//
FOR _i := GVL.PROG_CMDS_ARR_BEG TO GVL.PROG_CMDS_ARR_END BY 1 DO
	PersistentVars.Programs[11].Commands[_i].CommandType := DUT_CommandType.Disabled;
	PersistentVars.Programs[11].Commands[_i].CommandString := '';
END_FOR
PersistentVars.Programs[11].ProgramName := 'Make Me an Egg, Please';
PersistentVars.Programs[11].Commands[0].CommandType := DUT_CommandType.Disabled;
PersistentVars.Programs[11].Commands[0].CommandString := '';

//
FOR _i := GVL.PROG_CMDS_ARR_BEG TO GVL.PROG_CMDS_ARR_END BY 1 DO
	PersistentVars.Programs[12].Commands[_i].CommandType := DUT_CommandType.Disabled;
	PersistentVars.Programs[12].Commands[_i].CommandString := '';
END_FOR
PersistentVars.Programs[12].ProgramName := 'Egg Pick Routine';
PersistentVars.Programs[12].Commands[0].CommandType := DUT_CommandType.Disabled;
PersistentVars.Programs[12].Commands[0].CommandString := '';

//
FOR _i := GVL.PROG_CMDS_ARR_BEG TO GVL.PROG_CMDS_ARR_END BY 1 DO
	PersistentVars.Programs[13].Commands[_i].CommandType := DUT_CommandType.Disabled;
	PersistentVars.Programs[13].Commands[_i].CommandString := '';
END_FOR
PersistentVars.Programs[13].ProgramName := 'Egg Crack Routine';
PersistentVars.Programs[13].Commands[0].CommandType := DUT_CommandType.Disabled;
PersistentVars.Programs[13].Commands[0].CommandString := '';

//
FOR _i := GVL.PROG_CMDS_ARR_BEG TO GVL.PROG_CMDS_ARR_END BY 1 DO
	PersistentVars.Programs[14].Commands[_i].CommandType := DUT_CommandType.Disabled;
	PersistentVars.Programs[14].Commands[_i].CommandString := '';
END_FOR
PersistentVars.Programs[14].ProgramName := 'Egg Flip Routine';
PersistentVars.Programs[14].Commands[0].CommandType := DUT_CommandType.Disabled;
PersistentVars.Programs[14].Commands[0].CommandString := '';

//
FOR _i := GVL.PROG_CMDS_ARR_BEG TO GVL.PROG_CMDS_ARR_END BY 1 DO
	PersistentVars.Programs[15].Commands[_i].CommandType := DUT_CommandType.Disabled;
	PersistentVars.Programs[15].Commands[_i].CommandString := '';
END_FOR
PersistentVars.Programs[15].ProgramName := 'Egg Place Routine';
PersistentVars.Programs[15].Commands[0].CommandType := DUT_CommandType.Disabled;
PersistentVars.Programs[15].Commands[0].CommandString := '';
END_METHOD

METHOD M_Init : BOOL

// check if arfbot has been initialized
IF NOT PersistentVars.Flags[GVL.INIT_POS_IDX].Value THEN
	// poses
	PersistentVars.Flags[GVL.HOM_TO_POSE_IDX].Value := FALSE;
	PersistentVars.StoredPositions[GVL.POSE_1_IDX].Position.X := 0.0;
	PersistentVars.StoredPositions[GVL.POSE_1_IDX].Position.Y := -15.0;
	PersistentVars.StoredPositions[GVL.POSE_1_IDX].Position.Z := 115.0;
	PersistentVars.StoredPositions[GVL.POSE_1_IDX].Position.A := 0.0;
	PersistentVars.StoredPositions[GVL.POSE_1_IDX].Position.B := 30.0;
	PersistentVars.StoredPositions[GVL.POSE_1_IDX].Position.C := 0.0;
	
	PersistentVars.StoredPositions[GVL.POSE_2_IDX].Position.X := 0.0;
	PersistentVars.StoredPositions[GVL.POSE_2_IDX].Position.Y := -15.0;
	PersistentVars.StoredPositions[GVL.POSE_2_IDX].Position.Z := 115.0;
	PersistentVars.StoredPositions[GVL.POSE_2_IDX].Position.A := 0.0;
	PersistentVars.StoredPositions[GVL.POSE_2_IDX].Position.B := -30.0;
	PersistentVars.StoredPositions[GVL.POSE_2_IDX].Position.C := 0.0;
		 
	// decoder
	PersistentVars.StoredPositions[GVL.DEC_START_POS].Position.X := 300.0; // TODO need to verify all 6 of these
	PersistentVars.StoredPositions[GVL.DEC_START_POS].Position.Y := 0.0;
	PersistentVars.StoredPositions[GVL.DEC_START_POS].Position.Z := -400.0;
	PersistentVars.StoredPositions[GVL.DEC_START_POS].Position.A := 0.0;
	PersistentVars.StoredPositions[GVL.DEC_START_POS].Position.B := 0.0;
	PersistentVars.StoredPositions[GVL.DEC_START_POS].Position.C := 0.0;
	
	// set homing offsets
	PersistentVars.StoredPositions[GVL.HOM_POS_IDX].Position.X := 166; // J1 initial home offset
	PersistentVars.StoredPositions[GVL.HOM_POS_IDX].Position.Y := -35.3; // J2 initial home offset
	PersistentVars.StoredPositions[GVL.HOM_POS_IDX].Position.Z := 145; // J3 initial home offset
	PersistentVars.StoredPositions[GVL.HOM_POS_IDX].Position.A := -166; // J4 initial home offset
	PersistentVars.StoredPositions[GVL.HOM_POS_IDX].Position.B := -99.2; // J5 initial home offset
	PersistentVars.StoredPositions[GVL.HOM_POS_IDX].Position.C := 178; // J6 initial home offset
	
	// set speeds
	PersistentVars.StoredPositions[GVL.SPEEDS_IDX].Position.X := 100.0; // max velocity
	PersistentVars.StoredPositions[GVL.SPEEDS_IDX].Position.Y := 1000.0; // max accel/decel
	PersistentVars.StoredPositions[GVL.SPEEDS_IDX].Position.Z := 1000.0; // max jerk
	PersistentVars.StoredPositions[GVL.SPEEDS_IDX].Position.A := 1.0; // velocity factor
	PersistentVars.StoredPositions[GVL.SPEEDS_IDX].Position.B := 0.05; // accel/decel factor
	PersistentVars.StoredPositions[GVL.SPEEDS_IDX].Position.C := 1.0; // jerk factor
	
	//
	M_BuildTests();
		 
	// indicate initialized
	PersistentVars.Flags[GVL.INIT_POS_IDX].Value := TRUE;
END_IF

//
PersistentVars.StoredPositions[GVL.SPEEDS_IDX].Comment := 'vel, acc, jerk, vel fact, acc fact, jerk fact';
PersistentVars.StoredPositions[GVL.HOM_POS_IDX].Comment := 'Home Offsets J1, J2, J3, J4, J5, J6';
PersistentVars.StoredPositions[GVL.DEC_START_POS].Comment := 'NC Decoder Start Position';
PersistentVars.StoredPositions[GVL.TCP_POS_IDX].Comment := 'TCP Offset';
PersistentVars.StoredPositions[GVL.UC2_POS_IDX].Comment := 'UCS 2 Offset';
PersistentVars.StoredPositions[GVL.UC1_POS_IDX].Comment := 'UCS 1 Offset';
PersistentVars.StoredPositions[GVL.MCS_POS_IDX].Comment := 'MCS Offset';

//	 
PersistentVars.StoredPositions[GVL.POSE_1_IDX].Comment := 'Pose 1 coordinates';
PersistentVars.StoredPositions[GVL.POSE_2_IDX].Comment := 'Pose 2 coordinates';
PersistentVars.StoredPositions[GVL.POSE_3_IDX].Comment := 'Pose 3 coordinates';
PersistentVars.StoredPositions[GVL.POSE_4_IDX].Comment := 'Pose 4 coordinates';
PersistentVars.StoredPositions[GVL.POSE_5_IDX].Comment := 'Pose 5 coordinates';

//
PersistentVars.Flags[GVL.HOM_TO_POSE_IDX].Comment := 'Finish home at Pose';

//
PersistentVars.Flags[GVL.HOME_COMPLETE].Comment := 'Axes are homed';
PersistentVars.Flags[GVL.HOME_COMPLETE].Value := FALSE;

//
PersistentVars.Flags[GVL.INIT_POS_IDX].Comment := 'Variables are Intitialized';
END_METHOD

END_PROGRAM

// ---- FB/group/FB_GroupHandler.TcPOU
FUNCTION_BLOCK FB_GroupHandler
VAR CONSTANT
	NumberOfAxes: UINT:=GVL.NumberOfAxes;
END_VAR
VAR_IN_OUT
	AxisGroup: AXES_GROUP_REF;
	ACS: ARRAY[1..NumberOfAxes] OF AXIS_REF;
	MCS: ARRAY[1..NumberOfAxes] OF AXIS_REF;
END_VAR
VAR_INPUT
	Enable: BOOL;
	StoredPositions: REFERENCE TO ARRAY[GVL.POS_ARR_BEG..GVL.POS_ARR_END] OF DUT_StoredPosition;
END_VAR
VAR_OUTPUT
	Busy: BOOL;
	Error: BOOL;
	ErrorID: UDINT;
END_VAR
VAR
	
	_stKinToPlc     AT %I*     : NCTOPLC_NCICHANNEL_REF;
	_stPlcToKin     AT %Q*     : PLCTONC_NCICHANNEL_REF;
	
	//
	EnableFtrig: F_TRIG;
	
    _KinAxes: ST_KinAxes;
	
	//
	_SeqEnableGroup: INT;
	_SeqDisableGroup: INT;
	_SequenceSetKinematics: INT;
	_SequenceSetTrans: INT;
	_SeqResetGroup: INT;
	
	//
	_FB_AddAllAxes: FB_AddAllAxes;
	_FB_PowerAll: FB_PowerAll;
	_GroupPower: BOOL;
	_MC_GroupEnable: MC_GroupEnable;
	_MC_GroupStop: MC_GroupStop;
	_MC_UngroupAllAxes: MC_UngroupAllAxes;
	_MC_GroupDisable: MC_GroupDisable;
	_MC_GroupReset: MC_GroupReset;
	_FB_KinResetGroup: FB_KinResetGroup;
	_FB_KinCheckActualStatus: FB_KinCheckActualStatus;
    
    //
    _FB_KinConfigGroup: FB_KinConfigGroup;
	_McsCoordinateFrame: FB_CoordinateFrame;
	_Ucs1CoordinateFrame: FB_CoordinateFrame;
	_Ucs2CoordinateFrame: FB_CoordinateFrame;
	_TcpCoordinateFrame: FB_CoordinateFrame;
	_McsOffsetFrame: DUT_CoordFrame;
	_Ucs1OffsetFrame: DUT_CoordFrame;
	_Ucs2OffsetFrame: DUT_CoordFrame;
	_TcpOffsetFrame: DUT_CoordFrame;
	
	_MC_SetCoordinateTransform: MC_SetCoordinateTransform;
	_CoordinateSystem: DUT_CoordSystem;
	
	_GroupReady: BOOL;
	_EnableGroup: BOOL;
	_DisableGroup: BOOL;
	_GroupEnabled: BOOL;
	_ResetGroup: BOOL;
	_SetKinematics: BOOL;
	_SetCoordinates: BOOL;
	_KinematicsSet: BOOL;
	_CartesianMode: BOOL;
	_SetTransform: BOOL;
	_TransformSet: BOOL;
	
	_MC_GroupReadStatus: MC_GroupReadStatus;
	_DUT_GroupStatus: DUT_GroupStatus;
	
	_i, _j, _k: UINT;
	
END_VAR

VAR CONSTANT
	STEP_DONE: 				INT := 1000;
	STEP_IDLE: 				INT := 0000;
	STEP_GROUP_POWER_ON: 	INT := 0022;
	STEP_WAIT_POWER_ON: 	INT := 0024;
	STEP_GROUP_ENABLE: 		INT := 0030;
	STEP_WAIT_ENABLE: 		INT := 0035;
	STEP_READ_POSITION: 	INT := 0040;
	STEP_WAIT_POSITION: 	INT := 0050;
	STEP_SET_KINEMATICS: 	INT := 0060;
	STEP_WAIT_KINEMATICS: 	INT := 0070;
	STEP_SET_COORD_TRANS: 	INT := 0071;
	STEP_WAIT_COORD_TRANS: 	INT := 0072;
	STEP_GROUP_DISABLE: 	INT := 0100;
	STEP_WAIT_DISABLE: 		INT := 0110;
	STEP_GROUP_POWER_OFF: 	INT := 0120;
END_VAR

//
Busy := _SeqEnableGroup <> 0
		OR _SeqDisableGroup <> 0
		OR _SequenceSetKinematics <> 0
		OR _SequenceSetTrans <> 0
		OR _SeqResetGroup <> 0;
		
EnableFtrig(CLK:=Enable);
IF EnableFtrig.Q THEN
	M_DisableGroup();
END_IF

//
_M_EnableGroup();
_M_DisableGroup();
_M_SetKinematics();
_M_SetTransform();
_M_ResetGroup();

// https://infosys.beckhoff.com/content/1033/tf5240_kinematic_transformation/292852107.html?id=2424647827091372088
(* read the IDs from the cyclic axis interface so the axes can mapped later to the kinematic group *)
FOR _i:=1 TO NumberOfAxes BY 1 DO
	_KinAxes.nAxisIdsAcs[_i] := ACS[_i].NcToPlc.AxisId;
	_KinAxes.nAxisIdsMcs[_i] := MCS[_i].NcToPlc.AxisId;
END_FOR

//	
_FB_KinCheckActualStatus(
	bExecute:= , 
	stAxesListReference:= _KinAxes, 
	stKinRefIn:= _stKinToPlc, 
	eKinStatus=> ,
	bBusy=> , 
	bDone=> , 
	bError=> , 
	nErrorId=> );
	
// https://infosys.beckhoff.com/content/1033/tf5110-tf5113_tc3_kinematic_transformation/5737129739.html?id=6958083974342297833
// apparently we cannot use this for user specific transformations. dammit.
(*
_FB_KinCalcTrafo(
	bExecute:= , 
	bForward:= , 
	oidTrafo:= , // find object id in the General tab of the kinematic group
	stAxesPosIn:= , // if forward, these would be joint positions. if reverse, these would be cartesian
	stAxesPosOut:= , // if forward, these would be cartesian. if reverse, these would be joint positions
	uMetaInfoIn:= , 
	uMetaInfoOut:= , 
	bBusy=> , 
	bDone=> , 
	bError=> , 
	nErrorId=> );
*)

IF _CoordinateSystem = DUT_CoordSystem.ACS THEN
	_DUT_GroupStatus.CurrentPosition.X := ACS[1].NcToPlc.ActPos;
	_DUT_GroupStatus.CurrentPosition.Y := ACS[2].NcToPlc.ActPos;
	_DUT_GroupStatus.CurrentPosition.Z := ACS[3].NcToPlc.ActPos;
	_DUT_GroupStatus.CurrentPosition.A := ACS[4].NcToPlc.ActPos;
	_DUT_GroupStatus.CurrentPosition.B := ACS[5].NcToPlc.ActPos;
	_DUT_GroupStatus.CurrentPosition.C := ACS[6].NcToPlc.ActPos;
ELSE
	_DUT_GroupStatus.CurrentPosition.X := MCS[1].NcToPlc.ActPos;
	_DUT_GroupStatus.CurrentPosition.Y := MCS[2].NcToPlc.ActPos;
	_DUT_GroupStatus.CurrentPosition.Z := MCS[3].NcToPlc.ActPos;
	_DUT_GroupStatus.CurrentPosition.A := MCS[4].NcToPlc.ActPos;
	_DUT_GroupStatus.CurrentPosition.B := MCS[5].NcToPlc.ActPos;
	_DUT_GroupStatus.CurrentPosition.C := MCS[6].NcToPlc.ActPos;
END_IF

_MC_GroupReadStatus(
	AxesGroup:= AxisGroup, 
	Enable:= Enable, 
	Valid=> _DUT_GroupStatus.Valid, 
	Busy=> _DUT_GroupStatus.Busy, 
	GroupMoving=> _DUT_GroupStatus.GroupMoving, 
	GroupHoming=> _DUT_GroupStatus.GroupHoming, 
	GroupErrorStop=> _DUT_GroupStatus.GroupErrorStop, 
	GroupNotReady=> _DUT_GroupStatus.GroupNotReady, 
	GroupStandby=> _DUT_GroupStatus.GroupStandby, 
	GroupStopping=> _DUT_GroupStatus.GroupStopping, 
	GroupDisabled=> _DUT_GroupStatus.GroupDisabled, 
	AllAxesStanding=> _DUT_GroupStatus.AllAxesStanding, 
	InPosition=> _DUT_GroupStatus.InPosition, 
	Error=> _DUT_GroupStatus.Error, 
	ErrorId=> _DUT_GroupStatus.ErrorID);
	
_FB_PowerAll(
	Enable:= _GroupPower, 
	acs:= ACS, 
	mcs:= MCS, 
	Status=> , 
	Error=> );
	
_FB_KinConfigGroup(
	bExecute:= , 
	bCartesianMode:= , 
	stAxesList:= _KinAxes, 
	stKinRefIn:= _stKinToPlc, 
	bBusy=> , 
	bDone=> , 
	bError=> , 
	nErrorId=> );
	
_FB_AddAllAxes(
	Execute:= , 
	stGroupRef:= AxisGroup, 
	mcs:= MCS, 
	Done=> , 
	Busy=> , 
	Error=> );

_MC_GroupEnable(
	AxesGroup:= AxisGroup, 
	Execute:= , 
	Done=> , 
	Busy=> , 
	Error=> , 
	ErrorID=> );
	
_MC_GroupStop(
	AxesGroup:= AxisGroup, 
	Execute:= , 
	Deceleration:= , 
	Jerk:= MC_IGNORE, 
	Done=> , 
	Busy=> , 
	Active=> , 
	CommandAborted=> , 
	Error=> , 
	ErrorId=> );
	
_MC_UngroupAllAxes(
	AxesGroup:= AxisGroup, 
	Execute:= , 
	Done=> , 
	Busy=> , 
	Error=> , 
	ErrorId=> );
	
_MC_GroupDisable(
	AxesGroup:= AxisGroup, 
	Execute:= , 
	Done=> , 
	Busy=> , 
	Error=> , 
	ErrorID=> );

_FB_KinResetGroup(
	bExecute:= , 
	nItpChannelId:= , 
	stKinRefIn:= _stKinToPlc, 
	stAxesList:= _KinAxes, 
	bBusy=> , 
	bDone=> , 
	bError=> , 
	nErrorId=> );
	
_MC_GroupReset(
	AxesGroup:= AxisGroup, 
	Execute:= , 
	Done=> , 
	Busy=> , 
	Error=> , 
	ErrorId=> );
	
_McsCoordinateFrame(
	Execute:= , 
	oidTrafo:= GVL.McsCoordRef, 
	OffsetFrame:= _McsOffsetFrame, 
	Done=> , 
	Busy=> , 
	Error=> );
	
_Ucs1CoordinateFrame(
	Execute:= , 
	oidTrafo:= GVL.Ucs1CoordRef, 
	OffsetFrame:= _Ucs1OffsetFrame, 
	Done=> , 
	Busy=> , 
	Error=> );
	
_Ucs2CoordinateFrame(
	Execute:= , 
	oidTrafo:= GVL.Ucs2CoordRef, 
	OffsetFrame:= _Ucs2OffsetFrame, 
	Done=> , 
	Busy=> , 
	Error=> );
	
_TcpCoordinateFrame(
	Execute:= , 
	oidTrafo:= GVL.TcpCoordRef, 
	OffsetFrame:= _TcpOffsetFrame, 
	Done=> , 
	Busy=> , 
	Error=> );
	
_MC_SetCoordinateTransform(
	AxesGroup:= AxisGroup, 
	Execute:= , 
	CoordTransform:= , 
	Done=> , 
	Busy=> , 
	Active=> , 
	CommandAborted=> , 
	Error=> , 
	ErrorId=> );

METHOD PRIVATE _M_DisableGroup : BOOL

CASE _SeqDisableGroup OF
	0: // IDLE
		IF _DisableGroup THEN
			_DisableGroup := FALSE;
			_MC_UngroupAllAxes.Execute := FALSE;
			_MC_GroupDisable.Execute := FALSE;
			_MC_GroupEnable.Execute := FALSE;
			_MC_GroupReset.Execute := FALSE;
			_SeqDisableGroup := _SeqDisableGroup + 1;
		END_IF
		
	1:
		_MC_GroupDisable.Execute := TRUE;
		_SeqDisableGroup := _SeqDisableGroup + 1;
		
	2:
		// TODO add timeout timer here
		IF _MC_GroupDisable.Error THEN
			Error := TRUE;
			//ErrorID := ;
			_SeqDisableGroup := 0;
		ELSIF _MC_GroupDisable.Done THEN
			_MC_GroupDisable.Execute := FALSE;
			_SeqDisableGroup := _SeqDisableGroup + 1;
		END_IF
		
	3:
		_MC_UngroupAllAxes.Execute := TRUE;
		_SeqDisableGroup := _SeqDisableGroup + 1;
	
	4:
		IF _MC_UngroupAllAxes.Error THEN
			Error := TRUE;
			//ErrorID := ;
			_SeqDisableGroup := 0;
		ELSIF _MC_UngroupAllAxes.Done THEN
			_MC_UngroupAllAxes.Execute := FALSE;
			_SeqDisableGroup := _SeqDisableGroup + 1;
		END_IF
		
	5:
		_FB_KinResetGroup.bExecute := TRUE;
		_SeqDisableGroup := _SeqDisableGroup + 1;
		
	6:
		IF _FB_KinResetGroup.bDone OR _FB_KinResetGroup.bError
			OR _DUT_GroupStatus.GroupDisabled THEN
				_FB_KinResetGroup.bExecute := FALSE;
				_SeqDisableGroup := _SeqDisableGroup + 1;
		END_IF
	
	7:	
		_GroupReady := FALSE;
		_GroupEnabled := FALSE;
		_KinematicsSet := FALSE;
		_GroupPower := FALSE;
		_SeqDisableGroup := 0;
		
END_CASE
END_METHOD

METHOD PRIVATE _M_EnableGroup : BOOL

CASE _SeqEnableGroup OF
	0: // IDLE
		IF _EnableGroup THEN
			_EnableGroup := FALSE;
			_GroupEnabled := FALSE;
			_GroupReady := FALSE;
			_MC_GroupEnable.Execute := FALSE;
			_FB_AddAllAxes.Execute := FALSE;
			_SeqEnableGroup := _SeqEnableGroup + 1;
		END_IF
		
	1:
		_GroupPower := TRUE;
		_SeqEnableGroup := _SeqEnableGroup + 1;
		
	2:
		// TODO add timeout timer here
		IF _FB_PowerAll.Error THEN
			Error := TRUE;
			//ErrorID := _FB_PowerAll.ErrorID; // TODO get error ID
			_SeqEnableGroup := 0;
		ELSIF _FB_PowerAll.Status THEN
			_SeqEnableGroup := _SeqEnableGroup + 1;
		END_IF
		
	3: 
		IF M_SetKinematics(NOT (_CoordinateSystem = DUT_CoordSystem.ACS)) THEN
			_SeqEnableGroup := _SeqEnableGroup + 1;
		ELSE
			Error := TRUE;
			//ErrorID := _FB_PowerAll.ErrorID; // TODO get error ID
			_SeqEnableGroup := 0;
		END_IF
		
	4:	// TODO add timeout timer here
		IF Error THEN
			_SeqEnableGroup := 0;
		ELSIF _KinematicsSet THEN 
			_SeqEnableGroup := _SeqEnableGroup + 1;
		END_IF
		
	5:
		_FB_AddAllAxes.Execute := TRUE;
		_SeqEnableGroup := _SeqEnableGroup + 1;
		
	6:
		// TODO add timeout timer here
		IF _FB_AddAllAxes.Error THEN
			Error := TRUE;
			//ErrorID := _FB_AddAllAxes.ErrorID; // TODO get error ID
			_SeqEnableGroup := 0;
		ELSIF _FB_AddAllAxes.Done THEN
			_FB_AddAllAxes.Execute := FALSE;
			_SeqEnableGroup := _SeqEnableGroup + 1;
		END_IF
		
	7:
		_MC_GroupEnable.Execute := TRUE;
		_SeqEnableGroup := _SeqEnableGroup + 1;
		
	8:
		// TODO add timeout timer here
		IF _MC_GroupEnable.Error THEN
			Error := TRUE;
			//ErrorID := _MC_GroupEnable.ErrorID; // TODO get error ID
			_SeqEnableGroup := 0;
		ELSIF _MC_GroupEnable.Done THEN
			_GroupEnabled := TRUE;
			_SeqEnableGroup := _SeqEnableGroup + 1;
		END_IF;
		
	9:
		IF M_SetTransform(_CoordinateSystem) THEN
			_SeqEnableGroup := _SeqEnableGroup + 1;
		ELSE
			Error := TRUE;
			//ErrorID := ; // TODO get error ID
			_SeqEnableGroup := 0;
		END_IF
		
	10: 
		// TODO add timeout timer here
		IF Error THEN
			_SeqEnableGroup := 0;
		ELSIF _TransformSet THEN
			_GroupReady := TRUE;
			_SeqEnableGroup := 0;
		END_IF
		
END_CASE
END_METHOD

METHOD PRIVATE _M_ResetGroup : BOOL

CASE _SeqResetGroup OF
	0: // IDLE
		IF _ResetGroup THEN
			_ResetGroup := FALSE;
			//IF Error THEN // could do this for auto reset. commenting out for now.
				Error := FALSE;
				ErrorID := 0;
				_SeqResetGroup := _SeqResetGroup + 1;
			//END_IF
		END_IF
		
	1:
		IF NOT _DUT_GroupStatus.GroupDisabled THEN
			_FB_KinResetGroup.bExecute := TRUE;
		END_IF
		_SeqResetGroup := _SeqResetGroup + 1;
		
	2:
		IF _FB_KinResetGroup.bDone OR _FB_KinResetGroup.bError
			OR _DUT_GroupStatus.GroupDisabled THEN
				_FB_KinResetGroup.bExecute := FALSE;
				_SeqResetGroup := _SeqResetGroup + 1;
		END_IF
		
	3:
		_MC_GroupReset.Execute := TRUE;
		_SeqResetGroup := _SeqResetGroup + 1;
		
	4:
		IF _MC_GroupReset.Done OR _MC_GroupReset.Error THEN
			_MC_GroupReset.Execute := FALSE;
			_SeqResetGroup := _SeqResetGroup + 1;
		END_IF
	
	5: 
		//
		_SeqEnableGroup := 0;
		_SeqDisableGroup := 0;
		_SequenceSetKinematics := 0;
		_SequenceSetTrans := 0;
		_SeqResetGroup := 0;
	
END_CASE
END_METHOD

METHOD PRIVATE _M_SetKinematics : BOOL

CASE _SequenceSetKinematics OF
	0: // IDLE
		IF _SetKinematics THEN
			_SetKinematics := FALSE;
			_KinematicsSet := FALSE;
			_FB_KinConfigGroup.bExecute := FALSE;
			_SequenceSetKinematics := _SequenceSetKinematics + 1;
		END_IF
		
	1: // set kinematics
		_FB_KinConfigGroup.bExecute := TRUE;
		_FB_KinConfigGroup.bCartesianMode := _CartesianMode;
		_SequenceSetKinematics := _SequenceSetKinematics + 1;
		
	2: // wait for set kinematics
		// TODO add timeout timer here
		IF _FB_KinConfigGroup.bError THEN
			Error := TRUE;
			ErrorID := _FB_KinConfigGroup.nErrorId;
			_SequenceSetKinematics := 0;
		ELSIF _FB_KinConfigGroup.bDone THEN
			_FB_KinConfigGroup.bExecute := FALSE;
			_KinematicsSet := TRUE;
			_SequenceSetKinematics := 0;
		END_IF
		
END_CASE
END_METHOD

METHOD PRIVATE _M_SetTransform : BOOL
VAR_INPUT
END_VAR

CASE _SequenceSetTrans OF

	0: //
		IF _SetTransform THEN
			_SetTransform := FALSE;
			_TransformSet := FALSE;
			_McsCoordinateFrame.Execute := FALSE;
			_Ucs1CoordinateFrame.Execute := FALSE;
			_Ucs2CoordinateFrame.Execute := FALSE;
			_TcpCoordinateFrame.Execute := FALSE;
			_MC_SetCoordinateTransform.Execute := FALSE;
			_SequenceSetTrans := _SequenceSetTrans + 1;
		END_IF
		
	1: //
		_McsOffsetFrame.Position := StoredPositions[GVL.MCS_POS_IDX].Position;
		_McsOffsetFrame.Interpretation := MC.CoordInterpretation_SO3.Rotation_Z3Y2X1_DIN9300; // TODO make configurable
		_McsOffsetFrame.Direction := MC.ReferenceDefDir.fromReference; // TODO make configurable
		_McsCoordinateFrame.Execute := TRUE;
		
		_Ucs1OffsetFrame.Position := StoredPositions[GVL.UC1_POS_IDX].Position;
		_Ucs1OffsetFrame.Interpretation := MC.CoordInterpretation_SO3.Rotation_Z3Y2X1_DIN9300; // TODO make configurable
		_Ucs1OffsetFrame.Direction := MC.ReferenceDefDir.fromReference; // TODO make configurable
		_Ucs1CoordinateFrame.Execute := TRUE;
		
		_Ucs2OffsetFrame.Position := StoredPositions[GVL.UC2_POS_IDX].Position;
		_Ucs2OffsetFrame.Interpretation := MC.CoordInterpretation_SO3.Rotation_Z3Y2X1_DIN9300; // TODO make configurable
		_Ucs2OffsetFrame.Direction := MC.ReferenceDefDir.fromReference; // TODO make configurable
		_Ucs2CoordinateFrame.Execute := TRUE;
		
		// tcp will be set to the current mcs position plus any offset in the configuration
		_TcpOffsetFrame.Position.X := MCS[1].NcToPlc.ActPos + StoredPositions[GVL.TCP_POS_IDX].Position.X;
		_TcpOffsetFrame.Position.Y := MCS[2].NcToPlc.ActPos + StoredPositions[GVL.TCP_POS_IDX].Position.Y;
		_TcpOffsetFrame.Position.Z := MCS[3].NcToPlc.ActPos + StoredPositions[GVL.TCP_POS_IDX].Position.Z;
		_TcpOffsetFrame.Position.A := MCS[4].NcToPlc.ActPos + StoredPositions[GVL.TCP_POS_IDX].Position.A;
		_TcpOffsetFrame.Position.B := MCS[5].NcToPlc.ActPos + StoredPositions[GVL.TCP_POS_IDX].Position.B;
		_TcpOffsetFrame.Position.C := MCS[6].NcToPlc.ActPos + StoredPositions[GVL.TCP_POS_IDX].Position.C;
		//_TcpOffsetFrame.Position := StoredPositions[GVL.TCP_POS_IDX].Position;
		_TcpOffsetFrame.Interpretation := MC.CoordInterpretation_SO3.Rotation_Z3Y2X1_DIN9300; // TODO make configurable
		_TcpOffsetFrame.Direction := MC.ReferenceDefDir.fromReference; // TODO make configurable
		_TcpCoordinateFrame.Execute := TRUE;
		_SequenceSetTrans := _SequenceSetTrans + 1;
		
	2: //
		// TODO add timeout timer here
		IF _McsCoordinateFrame.Error
			OR _Ucs1CoordinateFrame.Error
			OR _Ucs2CoordinateFrame.Error
			OR _TcpCoordinateFrame.Error THEN
				(*SUPER^.M_Error(Description:=CONCAT('Move Command Error: ',
											CONCAT(TO_STRING(_MC_SetCoordinateTransform.ErrorID),
											CONCAT(' ', SMC_ErrorString(_MC_SetCoordinateTransform.ErrorID,
														SMC_Language_Type.english)))));*)
				//SUPER^.M_Error(Description:=CONCAT('Move Command Error: ', TO_STRING(_MC_SetCoordinateTransform.ErrorID)));
				_SequenceSetTrans := 10; // error step so we dont spam errors
			
		ELSIF _McsCoordinateFrame.Done 
				AND _Ucs1CoordinateFrame.Done 
				AND _Ucs2CoordinateFrame.Done 
				AND _TcpCoordinateFrame.Done THEN
					_McsCoordinateFrame.Execute := FALSE;
					_Ucs1CoordinateFrame.Execute := FALSE;
					_Ucs2CoordinateFrame.Execute := FALSE;
					_TcpCoordinateFrame.Execute := FALSE;
					_SequenceSetTrans := _SequenceSetTrans + 1;
		END_IF
		
	3:
		CASE _CoordinateSystem OF
			DUT_CoordSystem.ACS:
				_MC_SetCoordinateTransform.CoordTransform := GVL.McsCoordRef; // TODO: we shouldnt be here. maybe fault?
			DUT_CoordSystem.MCS:
				_MC_SetCoordinateTransform.CoordTransform := GVL.McsCoordRef;
			DUT_CoordSystem.UCS1:
				_MC_SetCoordinateTransform.CoordTransform := GVL.Ucs1CoordRef;
			DUT_CoordSystem.UCS2:
				_MC_SetCoordinateTransform.CoordTransform := GVL.Ucs2CoordRef;
			DUT_CoordSystem.TCP:
				_MC_SetCoordinateTransform.CoordTransform := GVL.TcpCoordRef;
		END_CASE
		_MC_SetCoordinateTransform.Execute := TRUE;
		_SequenceSetTrans := _SequenceSetTrans + 1;
	
	4: // wait for set coordinate transform
		// TODO add timeout timer here
		IF _MC_SetCoordinateTransform.Error THEN
			Error := TRUE;
			ErrorID := _MC_SetCoordinateTransform.ErrorID;
			_SequenceSetTrans := 0;
		ELSIF _MC_SetCoordinateTransform.Done THEN
			_TransformSet := TRUE;
			_SequenceSetTrans := 0;
		END_IF

END_CASE
END_METHOD

METHOD M_DisableGroup : BOOL
//IF NOT Error THEN
	M_DisableGroup := TRUE;
	_DisableGroup := TRUE;
//ELSE
	//M_DisableGroup := FALSE;
//END_IF
END_METHOD

METHOD M_EnableGroup : BOOL
VAR_INPUT
	CoordinateSystem: DUT_CoordSystem;
END_VAR
IF Enable (*AND NOT _GroupEnabled*) AND NOT Error THEN
	M_EnableGroup := TRUE;
	_CoordinateSystem := CoordinateSystem;
	_EnableGroup := TRUE;
	_GroupEnabled := FALSE;
ELSE
	M_EnableGroup := FALSE;
END_IF
END_METHOD

METHOD M_ResetGroup : BOOL
_ResetGroup := TRUE;
END_METHOD

METHOD PRIVATE M_SetKinematics : BOOL
VAR_INPUT
	CartesianMode: BOOL;
END_VAR
IF (_GroupEnabled OR _FB_PowerAll.Status) AND NOT Error THEN
	M_SetKinematics := TRUE;
	_SetKinematics := TRUE;
	_CartesianMode := CartesianMode;
	_KinematicsSet := FALSE;
ELSE
	M_SetKinematics := FALSE;
END_IF
END_METHOD

METHOD PUBLIC M_SetTransform : BOOL
VAR_INPUT
	CoordinateSystem: DUT_CoordSystem;
END_VAR
IF _GroupEnabled AND _KinematicsSet AND NOT Error THEN
	M_SetTransform := TRUE;
	_CoordinateSystem := CoordinateSystem;
	_SetTransform := TRUE;
	_TransformSet := FALSE;
ELSE
	M_SetTransform := FALSE;
END_IF
END_METHOD

{attribute 'monitoring' := 'variable'}
PROPERTY P_GroupReady : BOOL
GET
P_GroupReady := _GroupReady;
END_GET
END_PROPERTY

{attribute 'monitoring' := 'variable'}
PROPERTY P_GroupStatus : REFERENCE TO DUT_GroupStatus
GET
P_GroupStatus REF= _DUT_GroupStatus;
END_GET
END_PROPERTY

{attribute 'monitoring' := 'variable'}
PROPERTY P_KinematicsSet : BOOL
GET
P_KinematicsSet := _KinematicsSet;
END_GET
END_PROPERTY

{attribute 'monitoring' := 'variable'}
PROPERTY P_TransformSet : BOOL
GET
P_TransformSet := _TransformSet;
END_GET
END_PROPERTY

END_FUNCTION_BLOCK

// ---- FB/group/FB_AddAllAxes.TcPOU
FUNCTION_BLOCK FB_AddAllAxes
VAR_INPUT
	Execute				: BOOL;
END_VAR
VAR_IN_OUT
	stGroupRef: AXES_GROUP_REF;
	mcs: ARRAY[1..6] OF AXIS_REF;
END_VAR
VAR_OUTPUT
	Done				: BOOL;
	Busy				: BOOL;
	Error				: BOOL;
END_VAR
VAR
	fbAddAxis			: ARRAY[1..6] OF MC_AddAxisToGroup;
	i					: UINT;
END_VAR

Done := TRUE;
Busy := FALSE;
Error := FALSE;

// https://infosys.beckhoff.com/content/1033/tf5420_tc3_advanced_pick_and_place/8892979211.html?id=8490282963745653116
fbAddAxis[1].IdentInGroup := MCS_X; //X-Axis
fbAddAxis[2].IdentInGroup := MCS_Y; //Y-Axis
fbAddAxis[3].IdentInGroup := MCS_Z; //Z-Axis
fbAddAxis[4].IdentInGroup := ADDAX1; //MCS_A3;//
fbAddAxis[5].IdentInGroup := ADDAX2; //MCS_B2;//
fbAddAxis[6].IdentInGroup := ADDAX3; //MCS_C1;//

FOR i:=1 TO 6 DO
	fbAddAxis[i](AxesGroup:=stGroupRef, Axis := mcs[i], Execute := Execute);

	IF (NOT fbAddAxis[i].Done) THEN
		Done := FALSE;
	END_IF
	IF (fbAddAxis[i].Busy) THEN
		Busy := TRUE;
	END_IF
	IF (fbAddAxis[i].Error) THEN
		Error := TRUE;
	END_IF
END_FOR

END_FUNCTION_BLOCK

// ---- FB/coord/FB_CoordinateFrame.TcPOU
FUNCTION_BLOCK FB_CoordinateFrame
VAR_INPUT
	Execute: BOOL:=FALSE;
    oidTrafo: UDINT := 16#00000000; (*Trafo object id*)	
	OffsetFrame: DUT_CoordFrame:=(	Position:=(X:=0,Y:=0,Z:=0,A:=0,B:=0,C:=0),
									Interpretation:=MC.CoordInterpretation_SO3.Rotation_Z3Y2X1_DIN9300,
									Direction:=MC.ReferenceDefDir.fromReference);
END_VAR
VAR_OUTPUT
	Done: BOOL;
	Busy: BOOL;
	Error: BOOL;
END_VAR
VAR
	_ExecuteRtrig: R_TRIG;
	_ExecuteFtrig: F_TRIG;
	_DesiredOffset: ARRAY [1..6] OF LREAL;
	_fbKinUnlockTrafoParam: FB_KinUnlockTrafoParam;
	_fbKinLockTrafoParam: FB_KinLockTrafoParam;
	_LockParam, _UnlockParam : BOOL;
	_fbADSWRITE: ARRAY[1..8] OF ADSWRITE;
	_pidTrafo: ARRAY[1..8] OF UDINT := [16#05010110, 16#05010111, 16#05010112, 
										16#05010113, 16#05010114, 16#05010115,
										16#05010116, 16#05010117]; (*parameter id*)
	_i, _j, _k: INT;
	_Sequence: INT;
	_WriteDone, _WriteErr: BOOL;
END_VAR


// https://infosys.beckhoff.com/content/1033/tf5110-tf5113_tc3_kinematic_transformation/1955902347.html?id=3846917459939213436

_ExecuteRtrig(CLK:=Execute);
_ExecuteFtrig(CLK:=Execute);

IF _ExecuteFtrig.Q THEN
	_Sequence := 0;
	Error := FALSE;
	Done := FALSE;
	_UnlockParam := FALSE;
	_LockParam := FALSE;
END_IF

Busy := _Sequence <> 0;

CASE _Sequence OF
	0: // idle
		IF _ExecuteRtrig.Q THEN
			_Sequence := _Sequence + 1;
		END_IF
		
	1: // init
		Error := FALSE;
		Done := FALSE;
		_UnlockParam := FALSE;
		_LockParam := FALSE;
		_Sequence := _Sequence + 1;
		
	2: // unlock parameters
		_UnlockParam := TRUE;
		IF _fbKinUnlockTrafoParam.bDone THEN
			_Sequence := _Sequence + 1;
		ELSIF _fbKinUnlockTrafoParam.bError THEN
			_Sequence := 999;
		END_IF
		
	3: // 
		FOR _i := 1 TO 8 BY 1 DO
			_fbADSWRITE[_i](WRITE:=FALSE);
		END_FOR
		_DesiredOffset[1] := OffsetFrame.Position.X;
		_DesiredOffset[2] := OffsetFrame.Position.Y;
		_DesiredOffset[3] := OffsetFrame.Position.Z;
		_DesiredOffset[4] := OffsetFrame.Position.A;
		_DesiredOffset[5] := OffsetFrame.Position.B;
		_DesiredOffset[6] := OffsetFrame.Position.C;
		_Sequence := _Sequence + 1;
	
	4: // write parameters
		_WriteDone := TRUE;
		_WriteErr := FALSE;
		// write x, y, z, a, b, c
		FOR _i := 1 TO 6 BY 1 DO
			
			_fbADSWRITE[_i](PORT:=AMSPORT_R0_NCSAF, 
							IDXGRP:=oidTrafo, IDXOFFS:=_pidTrafo[_i], 
							LEN:=SIZEOF(_DesiredOffset[_i]), SRCADDR:=ADR(_DesiredOffset[_i]), 
							WRITE:=TRUE);
			IF _fbADSWRITE[_i].BUSY THEN
				_WriteDone := FALSE;
			ELSIF _fbADSWRITE[_i].ERR THEN
				_WriteErr := TRUE;
			END_IF
		END_FOR
		// write interpretation
		_i := 7;
		_fbADSWRITE[_i](PORT:=AMSPORT_R0_NCSAF, 
						IDXGRP:=oidTrafo, IDXOFFS:=_pidTrafo[_i], 
						LEN:=SIZEOF(OffsetFrame.Interpretation), SRCADDR:=ADR(OffsetFrame.Interpretation), 
						WRITE:=TRUE);
		IF _fbADSWRITE[_i].BUSY THEN
			_WriteDone := FALSE;
		ELSIF _fbADSWRITE[_i].ERR THEN
			_WriteErr := TRUE;
		END_IF
		// write direction
		_i := 8;
		_fbADSWRITE[_i](PORT:=AMSPORT_R0_NCSAF, 
						IDXGRP:=oidTrafo, IDXOFFS:=_pidTrafo[_i], 
						LEN:=SIZEOF(OffsetFrame.Direction), SRCADDR:=ADR(OffsetFrame.Direction), 
						WRITE:=TRUE);
		IF _fbADSWRITE[_i].BUSY THEN
			_WriteDone := FALSE;
		ELSIF _fbADSWRITE[_i].ERR THEN
			_WriteErr := TRUE;
		END_IF
		// go to next
		IF _WriteDone THEN
			_Sequence := _Sequence + 1;
		ELSIF _WriteErr THEN
			_Sequence := 999;
		END_IF
	
	5: // lock parameters
		_LockParam := TRUE;
		IF _fbKinLockTrafoParam.bDone THEN
			_Sequence := _Sequence + 1;
		ELSIF _fbKinLockTrafoParam.bError THEN
			_Sequence := 999;
		END_IF
	
	6: // done
		Done := TRUE;
		_Sequence := 0;
	
	999..9999: // error
		Error := TRUE;
	
END_CASE

_fbKinUnlockTrafoParam(
	bExecute:= _UnlockParam, 
	oidTrafo:= oidTrafo, 
	bBusy=> , 
	bDone=> , 
	bError=> , 
	nErrorId=> );
	
_fbKinLockTrafoParam(
	bExecute:= _LockParam, 
	oidTrafo:= oidTrafo, 
	bBusy=> , 
	bDone=> , 
	bError=> , 
	nErrorId=> );

END_FUNCTION_BLOCK

// ---- FB/home/FB_HomingProcessor.TcPOU
FUNCTION_BLOCK FB_HomingProcessor
VAR CONSTANT
	NumberOfAxes: UINT:=GVL.NumberOfAxes;
END_VAR
VAR_IN_OUT
	ACS: ARRAY[1..NumberOfAxes] OF AXIS_REF;
	AxisGroup: AXES_GROUP_REF;
	GroupHandler: FB_GroupHandler;
	//Controller: FB_Controller;
END_VAR
VAR_INPUT
	Enable: BOOL;
	Reset: BOOL;
	StoredPositions: REFERENCE TO ARRAY[GVL.POS_ARR_BEG..GVL.POS_ARR_END] OF DUT_StoredPosition;
	VisionRegisters: REFERENCE TO ARRAY[GVL.VIS_ARR_BEG..GVL.VIS_ARR_END] OF DUT_VisionRegister;
	Flags: REFERENCE TO ARRAY[GVL.FLG_ARR_BEG..GVL.FLG_ARR_END] OF DUT_Flags;
END_VAR
VAR_OUTPUT
	Done: BOOL;
	Busy: BOOL;
	Error: BOOL;
	ErrorID: UDINT;
END_VAR
VAR
	_ExecuteRtrig: R_TRIG;
	_ExecuteFtrig: F_TRIG;
	_ResetRtrig: R_TRIG;
	_ErrorRtrig: R_TRIG;
	
	_SequenceMain: INT;
	_StartHoming: BOOL;
	
	_SMC_Homing_J1, _SMC_Homing_J2, _SMC_Homing_J3: MC_Home;
	_SMC_Homing_J4, _SMC_Homing_J5, _SMC_Homing_J6: MC_Home;
    _ST_HomingOptions_J1,_ST_HomingOptions_J2,_ST_HomingOptions_J3: ST_HomingOptions;
    _ST_HomingOptions_J4,_ST_HomingOptions_J5,_ST_HomingOptions_J6: ST_HomingOptions;
	
	_MC_SetPosition_J1, _MC_SetPosition_J2, _MC_SetPosition_J3: MC_SetPosition;
	_MC_SetPosition_J4, _MC_SetPosition_J5, _MC_SetPosition_J6: MC_SetPosition;
    _ST_SetPositionsOptions_J1,_ST_SetPositionsOptions_J2,_ST_SetPositionsOptions_J3: ST_SetPositionOptions;
    _ST_SetPositionsOptions_J4,_ST_SetPositionsOptions_J5,_ST_SetPositionsOptions_J6: ST_SetPositionOptions;
	
	_HomingVelocityFast: LREAL:= 10.0;
	_HomingVelocitySlow: LREAL:= 5.0;
	_HomingVelocitySlowSlow: LREAL:= 1.0;
	_HomingAcceleration: LREAL:= 1000.0;
	_HomingJerk: LREAL:= 10000.0;
	
	_MoveToPose: BOOL;
	_MoveCommand: ST_MoveCmd;
	_MoveCommandProcessor: MoveCmdProcessor;
	
	_MC_MoveAbsolute: ARRAY[1..NumberOfAxes] OF MC_MoveAbsolute;
	
	_i, _j, _k: UINT;
	_FirstScan: BOOL:=TRUE;
END_VAR

VAR CONSTANT
	STEP_DONE: 					INT := 9999;
	STEP_IDLE: 					INT := 0000;
	STEP_GROUP_ENABLE: 			INT := 0030;
	STEP_WAIT_ENABLE: 			INT := 0035;
	STEP_FAST_HOME_G1:			INT := 0040;
	STEP_WAIT_FAST_HOME_G1:		INT := 0045;
	STEP_SLOW_HOME_G1:			INT := 0050;
	STEP_WAIT_SLOW_HOME_G1:		INT := 0055;
	STEP_MOVE_HOME_G1:			INT := 0056;
	
	STEP_FAST_HOME_G2:			INT := 0060;
	STEP_WAIT_FAST_HOME_G2:		INT := 0065;
	STEP_SLOW_HOME_G2:			INT := 0070;
	STEP_WAIT_SLOW_HOME_G2:		INT := 0075;
	STEP_MOVE_HOME_G2:			INT := 0076;
	
	STEP_FAST_HOME_G3:			INT := 0080;
	STEP_WAIT_FAST_HOME_G3:		INT := 0085;
	STEP_SLOW_HOME_G3:			INT := 0090;
	STEP_WAIT_SLOW_HOME_G3:		INT := 0095;
	STEP_MOVE_HOME_G3:			INT := 0096;
	
	STEP_MOVE_TO_POSE:			INT := 1000;
	STEP_WAIT_MOVE_TO_POSE:		INT := 1010;
	STEP_WAIT_POSE_DONE:		INT := 1020;
END_VAR

_ExecuteRtrig(CLK:=);
_ExecuteFtrig(CLK:=);
_ResetRtrig(CLK:=Reset);

IF _FirstScan THEN
	//
END_IF

CASE _SequenceMain OF
	STEP_DONE: // done
		Busy := FALSE;
		Done := TRUE;
		//_MoveCommandProcessor.M_Home();
		_SequenceMain := STEP_IDLE;
		
		_SMC_Homing_J1.Execute := FALSE;
		_SMC_Homing_J2.Execute := FALSE;
		_SMC_Homing_J3.Execute := FALSE;
		_SMC_Homing_J4.Execute := FALSE;
		_SMC_Homing_J5.Execute := FALSE;
		_SMC_Homing_J6.Execute := FALSE;
		
	STEP_IDLE: // IDLE
		IF _StartHoming AND Enable THEN
			_StartHoming := FALSE;
			Busy := TRUE;
			Done := FALSE;
			_SequenceMain := STEP_GROUP_ENABLE;
			Flags[GVL.HOME_COMPLETE].Value := FALSE;
		END_IF
		
	STEP_GROUP_ENABLE:
		IF GroupHandler.M_EnableGroup(DUT_CoordSystem.ACS) THEN
			_SequenceMain := STEP_WAIT_ENABLE;
		ELSE
			_SequenceMain := STEP_DONE;
			Error := TRUE;
			ErrorID := GroupHandler.ErrorID;
		END_IF
		
	STEP_WAIT_ENABLE:
		// TODO add timeout timer here
		IF GroupHandler.P_GroupReady THEN
			_SequenceMain := STEP_FAST_HOME_G1;
		END_IF;
		
	STEP_FAST_HOME_G1:	
		_SMC_Homing_J1.Execute := TRUE;
		_SMC_Homing_J2.Execute := TRUE;
		_SMC_Homing_J3.Execute := TRUE;
		_ST_HomingOptions_J1.SearchVelocity := _HomingVelocitySlow;
		_ST_HomingOptions_J2.SearchVelocity := _HomingVelocitySlow;
		_ST_HomingOptions_J3.SearchVelocity := _HomingVelocitySlow;
		_ST_HomingOptions_J1.SearchDirection := Tc2_MC2.MC_Direction.MC_Positive_Direction;
		_ST_HomingOptions_J2.SearchDirection := Tc2_MC2.MC_Direction.MC_Negative_Direction;
		_ST_HomingOptions_J3.SearchDirection := Tc2_MC2.MC_Direction.MC_Positive_Direction;
		_SequenceMain := STEP_WAIT_FAST_HOME_G1;
		
	STEP_WAIT_FAST_HOME_G1: // wait fast home group 1
		IF _SMC_Homing_J1.Done
			AND _SMC_Homing_J2.Done
			AND _SMC_Homing_J3.Done THEN
				_SMC_Homing_J1.Execute := FALSE;
				_SMC_Homing_J2.Execute := FALSE;
				_SMC_Homing_J3.Execute := FALSE;
				_SequenceMain := STEP_SLOW_HOME_G1;
		END_IF
		
	STEP_SLOW_HOME_G1: // slow home group 1
		_SMC_Homing_J1.Execute := TRUE;
		_SMC_Homing_J2.Execute := TRUE;
		_SMC_Homing_J3.Execute := TRUE;
		_ST_HomingOptions_J1.SearchVelocity := _HomingVelocitySlowSlow;
		_ST_HomingOptions_J2.SearchVelocity := _HomingVelocitySlow;
		_ST_HomingOptions_J3.SearchVelocity := _HomingVelocitySlowSlow;
		_SequenceMain := STEP_WAIT_SLOW_HOME_G1;
		
	STEP_WAIT_SLOW_HOME_G1:
		IF _SMC_Homing_J1.Done
			AND _SMC_Homing_J2.Done
			AND _SMC_Homing_J3.Done THEN
				_SMC_Homing_J1.Execute := FALSE;
				_SMC_Homing_J2.Execute := FALSE;
				_SMC_Homing_J3.Execute := FALSE;
				_MC_MoveAbsolute[1].Execute := FALSE;
				_MC_MoveAbsolute[2].Execute := FALSE;
				_MC_MoveAbsolute[3].Execute := FALSE;
				_SequenceMain := STEP_MOVE_HOME_G1;
		END_IF
		
	STEP_MOVE_HOME_G1:
		_MC_MoveAbsolute[1].Execute := TRUE;
		_MC_MoveAbsolute[2].Execute := TRUE;
		_MC_MoveAbsolute[3].Execute := TRUE;
		IF _MC_MoveAbsolute[1].Done 
			AND _MC_MoveAbsolute[2].Done 
			AND _MC_MoveAbsolute[3].Done THEN
				_SequenceMain := STEP_FAST_HOME_G2;
		END_IF
		
	STEP_FAST_HOME_G2:		
		_SMC_Homing_J4.Execute := TRUE;
		_SMC_Homing_J5.Execute := TRUE;
		_ST_HomingOptions_J4.SearchVelocity := _HomingVelocitySlow;
		_ST_HomingOptions_J5.SearchVelocity := _HomingVelocitySlow;
		_ST_HomingOptions_J4.SearchDirection := Tc2_MC2.MC_Direction.MC_Negative_Direction;
		_ST_HomingOptions_J5.SearchDirection := Tc2_MC2.MC_Direction.MC_Negative_Direction;
		_SequenceMain := STEP_WAIT_FAST_HOME_G2;
		
	STEP_WAIT_FAST_HOME_G2:
		IF _SMC_Homing_J4.Done
			AND _SMC_Homing_J5.Done THEN
				_SMC_Homing_J4.Execute := FALSE;
				_SMC_Homing_J5.Execute := FALSE;
				_SequenceMain := STEP_SLOW_HOME_G2;
		END_IF
		
	STEP_SLOW_HOME_G2:
		_SMC_Homing_J4.Execute := TRUE;
		_SMC_Homing_J5.Execute := TRUE;
		_ST_HomingOptions_J4.SearchVelocity := _HomingVelocitySlowSlow;
		_ST_HomingOptions_J5.SearchVelocity := _HomingVelocitySlowSlow;
		_SequenceMain := STEP_WAIT_SLOW_HOME_G2;
		
	STEP_WAIT_SLOW_HOME_G2:
		IF _SMC_Homing_J4.Done
			AND _SMC_Homing_J5.Done THEN
				_SMC_Homing_J4.Execute := FALSE;
				_SMC_Homing_J5.Execute := FALSE;
				_MC_MoveAbsolute[4].Execute := FALSE;
				_MC_MoveAbsolute[5].Execute := FALSE;
				_SequenceMain := STEP_MOVE_HOME_G2;
		END_IF
		
	STEP_MOVE_HOME_G2:
		_MC_MoveAbsolute[4].Execute := TRUE;
		_MC_MoveAbsolute[5].Execute := TRUE;
		IF _MC_MoveAbsolute[4].Done 
			AND _MC_MoveAbsolute[5].Done THEN
				_SequenceMain := STEP_FAST_HOME_G3;
		END_IF
		
	STEP_FAST_HOME_G3:
		_SMC_Homing_J6.Execute := TRUE;
		_ST_HomingOptions_J6.SearchVelocity := _HomingVelocitySlow;
		_ST_HomingOptions_J6.SearchDirection := Tc2_MC2.MC_Direction.MC_Positive_Direction;
		_SequenceMain := STEP_WAIT_FAST_HOME_G3;
		
	STEP_WAIT_FAST_HOME_G3:
		IF _SMC_Homing_J6.Done THEN
			_SMC_Homing_J6.Execute := FALSE;
			_SequenceMain := STEP_SLOW_HOME_G3;
		END_IF
		
	STEP_SLOW_HOME_G3:
		_SMC_Homing_J6.Execute := TRUE;
		_ST_HomingOptions_J6.SearchVelocity := _HomingVelocitySlowSlow;
		_SequenceMain := STEP_WAIT_SLOW_HOME_G3;
		
	STEP_WAIT_SLOW_HOME_G3:
		IF _SMC_Homing_J6.Done THEN
			_SMC_Homing_J6.Execute := FALSE;
			_MC_MoveAbsolute[6].Execute := FALSE;
			_SequenceMain := STEP_MOVE_HOME_G3;
		END_IF;
		
	STEP_MOVE_HOME_G3:
		_MC_MoveAbsolute[6].Execute := TRUE;
		IF _MC_MoveAbsolute[6].Done  THEN
			Flags[GVL.HOME_COMPLETE].Value := TRUE;
			IF NOT Flags[GVL.HOM_TO_POSE_IDX].Value THEN
				_SequenceMain := STEP_DONE;
			ELSE
				_SequenceMain := STEP_MOVE_TO_POSE;
			END_IF
		END_IF
		
	STEP_MOVE_TO_POSE:
		_MoveToPose := TRUE;
		_SequenceMain := STEP_WAIT_MOVE_TO_POSE;
	
	STEP_WAIT_MOVE_TO_POSE:
		IF _MoveCommandProcessor.ItfUnitMode.CurrentState <> PACK_ML.State.Idle THEN
			_SequenceMain := STEP_WAIT_POSE_DONE;
		END_IF
		
	STEP_WAIT_POSE_DONE:
		IF _MoveCommandProcessor.ItfUnitMode.CurrentState = PACK_ML.State.Idle THEN
			_SequenceMain := STEP_DONE;
		END_IF
	
END_CASE

_M_HandlePose();

//
IF _ResetRtrig.Q (*AND Error*) THEN
	Error := FALSE;
	ErrorID := 0;
	_SequenceMain := STEP_DONE;
	GroupHandler.M_ResetGroup();
	_MoveCommandProcessor.M_Home();
END_IF

//
_ErrorRtrig(CLK:=GroupHandler.Error
				OR _SMC_Homing_J1.Error
				OR _SMC_Homing_J2.Error
				OR _SMC_Homing_J3.Error
				OR _SMC_Homing_J4.Error
				OR _SMC_Homing_J5.Error
				OR _SMC_Homing_J6.Error
				OR _MoveCommandProcessor.Error);			
IF _ErrorRtrig.Q THEN
	Error := TRUE;
	IF GroupHandler.Error THEN
		ErrorID := GroupHandler.ErrorID;
	ELSIF _SMC_Homing_J1.Error THEN
		ErrorID := _SMC_Homing_J1.ErrorID;
	ELSIF _SMC_Homing_J2.Error THEN
		ErrorID := _SMC_Homing_J2.ErrorID;
	ELSIF _SMC_Homing_J3.Error THEN
		ErrorID := _SMC_Homing_J3.ErrorID;
	ELSIF _SMC_Homing_J4.Error THEN
		ErrorID := _SMC_Homing_J4.ErrorID;
	ELSIF _SMC_Homing_J5.Error THEN
		ErrorID := _SMC_Homing_J5.ErrorID;
	ELSIF _SMC_Homing_J6.Error THEN
		ErrorID := _SMC_Homing_J6.ErrorID;
	ELSIF _MoveCommandProcessor.Error THEN
		// TODO need to rework how error messages are handled (globally)
		// if the move command processor has an error, we dont know what it is.
	END_IF
END_IF

// https://infosys.beckhoff.com/content/1033/tcplclibmc2/458433931.html?id=4042515396221059782
//_ST_HomingOptions_J1.SearchDirection := MC_Negative_Direction;
_SMC_Homing_J1(
	Axis:= ACS[1], 
	Execute:= , 
	Position:=StoredPositions[GVL.HOM_POS_IDX].Position.X, // DEFAULT_HOME_POSITION, 
	HomingMode:= MC_HomingMode.MC_DefaultHoming, 
	BufferMode:= , 
	Options:= _ST_HomingOptions_J1, 
	bCalibrationCam:= , 
	Done=> , 
	Busy=> , 
	Active=> , 
	CommandAborted=> , 
	Error=> , 
	ErrorID=> );
_SMC_Homing_J2(
	Axis:= ACS[2], 
	Execute:= , 
	Position:=StoredPositions[GVL.HOM_POS_IDX].Position.Y, // DEFAULT_HOME_POSITION, 
	HomingMode:= MC_HomingMode.MC_DefaultHoming, 
	BufferMode:= , 
	Options:= _ST_HomingOptions_J2, 
	bCalibrationCam:= , 
	Done=> , 
	Busy=> , 
	Active=> , 
	CommandAborted=> , 
	Error=> , 
	ErrorID=> );
_SMC_Homing_J3(
	Axis:= ACS[3], 
	Execute:= , 
	Position:=StoredPositions[GVL.HOM_POS_IDX].Position.Z, // DEFAULT_HOME_POSITION, 
	HomingMode:= MC_HomingMode.MC_DefaultHoming, 
	BufferMode:= , 
	Options:= _ST_HomingOptions_J3, 
	bCalibrationCam:= , 
	Done=> , 
	Busy=> , 
	Active=> , 
	CommandAborted=> , 
	Error=> , 
	ErrorID=> );
_SMC_Homing_J4(
	Axis:= ACS[4], 
	Execute:= , 
	Position:=StoredPositions[GVL.HOM_POS_IDX].Position.A, // DEFAULT_HOME_POSITION, 
	HomingMode:= MC_HomingMode.MC_DefaultHoming, 
	BufferMode:= , 
	Options:= _ST_HomingOptions_J4, 
	bCalibrationCam:= , 
	Done=> , 
	Busy=> , 
	Active=> , 
	CommandAborted=> , 
	Error=> , 
	ErrorID=> );
_SMC_Homing_J5(
	Axis:= ACS[5], 
	Execute:= , 
	Position:=StoredPositions[GVL.HOM_POS_IDX].Position.B, // DEFAULT_HOME_POSITION, 
	HomingMode:= MC_HomingMode.MC_DefaultHoming, 
	BufferMode:= , 
	Options:= _ST_HomingOptions_J5, 
	bCalibrationCam:= , 
	Done=> , 
	Busy=> , 
	Active=> , 
	CommandAborted=> , 
	Error=> , 
	ErrorID=> );
_SMC_Homing_J6(
	Axis:= ACS[6], 
	Execute:= , 
	Position:=StoredPositions[GVL.HOM_POS_IDX].Position.C, // DEFAULT_HOME_POSITION, 
	HomingMode:= MC_HomingMode.MC_DefaultHoming, 
	BufferMode:= , 
	Options:= _ST_HomingOptions_J6, 
	bCalibrationCam:= , 
	Done=> , 
	Busy=> , 
	Active=> , 
	CommandAborted=> , 
	Error=> , 
	ErrorID=> );
	
//
_ST_SetPositionsOptions_J1.ClearPositionLag := TRUE;
_MC_SetPosition_J1(
	Axis:= ACS[1], 
	Execute:= _MC_SetPosition_J1.Execute AND NOT _MC_SetPosition_J1.Done AND NOT _MC_SetPosition_J1.Error, 
	Position:= 0.0, 
	Mode:= FALSE, // true=relative false=absolute
    Options:= _ST_SetPositionsOptions_J1,
	Done=> , 
	Busy=> , 
	Error=> , 
	ErrorID=> );
_ST_SetPositionsOptions_J2.ClearPositionLag := TRUE;
_MC_SetPosition_J2(
	Axis:= ACS[2], 
	Execute:= _MC_SetPosition_J2.Execute AND NOT _MC_SetPosition_J2.Done AND NOT _MC_SetPosition_J2.Error, 
	Position:= 0.0, 
	Mode:= FALSE, // true=relative false=absolute
    Options:= _ST_SetPositionsOptions_J2,
	Done=> , 
	Busy=> , 
	Error=> , 
	ErrorID=> );
_ST_SetPositionsOptions_J3.ClearPositionLag := TRUE;
_MC_SetPosition_J3(
	Axis:= ACS[3], 
	Execute:= _MC_SetPosition_J3.Execute AND NOT _MC_SetPosition_J3.Done AND NOT _MC_SetPosition_J3.Error, 
	Position:= 0.0, 
	Mode:= FALSE, // true=relative false=absolute
    Options:= _ST_SetPositionsOptions_J3,
	Done=> , 
	Busy=> , 
	Error=> , 
	ErrorID=> );
_ST_SetPositionsOptions_J4.ClearPositionLag := TRUE;
_MC_SetPosition_J4(
	Axis:= ACS[4], 
	Execute:= _MC_SetPosition_J4.Execute AND NOT _MC_SetPosition_J4.Done AND NOT _MC_SetPosition_J4.Error, 
	Position:= 0.0, 
	Mode:= FALSE, // true=relative false=absolute
    Options:= _ST_SetPositionsOptions_J4,
	Done=> , 
	Busy=> , 
	Error=> , 
	ErrorID=> );
_ST_SetPositionsOptions_J5.ClearPositionLag := TRUE;
_MC_SetPosition_J5(
	Axis:= ACS[5], 
	Execute:= _MC_SetPosition_J5.Execute AND NOT _MC_SetPosition_J5.Done AND NOT _MC_SetPosition_J5.Error, 
	Position:= 0.0, 
	Mode:= FALSE, // true=relative false=absolute
    Options:= _ST_SetPositionsOptions_J5,
	Done=> , 
	Busy=> , 
	Error=> , 
	ErrorID=> );
_ST_SetPositionsOptions_J6.ClearPositionLag := TRUE;
_MC_SetPosition_J6(
	Axis:= ACS[6], 
	Execute:= _MC_SetPosition_J6.Execute AND NOT _MC_SetPosition_J6.Done AND NOT _MC_SetPosition_J6.Error, 
	Position:= 0.0, 
	Mode:= FALSE, // true=relative false=absolute
    Options:= _ST_SetPositionsOptions_J6,
	Done=> , 
	Busy=> , 
	Error=> , 
	ErrorID=> );
	
FOR _k:= 1 TO NumberOfAxes DO
	_MC_MoveAbsolute[_k](
		Axis:= ACS[_k], 
		Execute:= , 
		Position:= 0.0, 
		Velocity:= _HomingVelocityFast, 
		Acceleration:= MC_DEFAULT, 
		Deceleration:= MC_DEFAULT, 
		Jerk:= MC_DEFAULT, 
		BufferMode:= , 
		Options:= , 
		Done=> , 
		Busy=> , 
		Active=> , 
		CommandAborted=> , 
		Error=> , 
		ErrorID=> );
END_FOR

METHOD PRIVATE _M_HandlePose : BOOL
VAR
	_MoveCommand: ST_MoveCmd;
	_PoseSpeed: LREAL := 20.0;
END_VAR
IF _MoveToPose THEN
	_MoveToPose:= FALSE;
	//
	IF GVL.PowerOn 
		AND_THEN Flags[GVL.HOME_COMPLETE].Value
		AND_THEN NOT _MoveCommandProcessor.Busy
		AND_THEN NOT _MoveCommandProcessor.Error THEN
			//
			_MoveCommand.MoveType 			:= DUT_Command_MoveType.DirectMove;
			_MoveCommand.PositionType 		:= DUT_Command_PositionType.AbsolutePosition;
			_MoveCommand.CoordinateType 	:= DUT_Command_CoordinateType.Literal;
			_MoveCommand.Speed 				:= _PoseSpeed;
			_MoveCommand.CoordSystem 		:= DUT_CoordSystem.ACS;
			_MoveCommand.CoordRef 			:= StoredPositions[GVL.POSE_2_IDX].Position;
			//
			_MoveCommandProcessor.Command := BuildMoveCmd(_MoveCommand);
			_MoveCommandProcessor.M_Start();
	END_IF;
END_IF

_MoveCommandProcessor(
	StoredPositions:= StoredPositions,
	VisionRegisters:= VisionRegisters,
	Flags:= Flags,
	AxisGroup:= AxisGroup, 
	GroupHandler:= GroupHandler,
	Velocity:= StoredPositions[GVL.SPEEDS_IDX].Position.X, 
	VelFactor:= StoredPositions[GVL.SPEEDS_IDX].Position.A,
	Acceleration:= StoredPositions[GVL.SPEEDS_IDX].Position.Y, 
	AccFactor:= StoredPositions[GVL.SPEEDS_IDX].Position.B,
	Jerk:= StoredPositions[GVL.SPEEDS_IDX].Position.Z,
	JerkFactor:= StoredPositions[GVL.SPEEDS_IDX].Position.C, 
	Position=> ,
	ItfUnitMode=> , 
	Error=> );
END_METHOD

METHOD M_SetHome : BOOL

// adjust all the persistent variables to take on the calibrated values
StoredPositions[GVL.HOM_POS_IDX].Position.X := F_HomeOffsetCalc(	CurrentOffset:= PersistentVars.StoredPositions[GVL.HOM_POS_IDX].Position.X, 
																				CurrentPosition:= ACS[1].NcToPlc.ActPos, 
																				HomeSearchDirection:= _ST_HomingOptions_J1.SearchDirection);

StoredPositions[GVL.HOM_POS_IDX].Position.Y := F_HomeOffsetCalc(	CurrentOffset:= PersistentVars.StoredPositions[GVL.HOM_POS_IDX].Position.Y, 
																				CurrentPosition:= ACS[2].NcToPlc.ActPos, 
																				HomeSearchDirection:= _ST_HomingOptions_J2.SearchDirection);

StoredPositions[GVL.HOM_POS_IDX].Position.Z := F_HomeOffsetCalc(	CurrentOffset:= PersistentVars.StoredPositions[GVL.HOM_POS_IDX].Position.Z, 
																				CurrentPosition:= ACS[3].NcToPlc.ActPos, 
																				HomeSearchDirection:= _ST_HomingOptions_J3.SearchDirection);

StoredPositions[GVL.HOM_POS_IDX].Position.A := F_HomeOffsetCalc(	CurrentOffset:= PersistentVars.StoredPositions[GVL.HOM_POS_IDX].Position.A, 
																				CurrentPosition:= ACS[4].NcToPlc.ActPos, 
																				HomeSearchDirection:= _ST_HomingOptions_J4.SearchDirection);

StoredPositions[GVL.HOM_POS_IDX].Position.B := F_HomeOffsetCalc(	CurrentOffset:= PersistentVars.StoredPositions[GVL.HOM_POS_IDX].Position.B, 
																				CurrentPosition:= ACS[5].NcToPlc.ActPos, 
																				HomeSearchDirection:= _ST_HomingOptions_J5.SearchDirection);

StoredPositions[GVL.HOM_POS_IDX].Position.C := F_HomeOffsetCalc(	CurrentOffset:= PersistentVars.StoredPositions[GVL.HOM_POS_IDX].Position.C, 
																				CurrentPosition:= ACS[6].NcToPlc.ActPos, 
																				HomeSearchDirection:= _ST_HomingOptions_J6.SearchDirection);

// this isnt totally needed but will calibrate the current session without the need to rehome
_MC_SetPosition_J1.Execute:=TRUE;
_MC_SetPosition_J2.Execute:=TRUE;
_MC_SetPosition_J3.Execute:=TRUE;
_MC_SetPosition_J4.Execute:=TRUE;
_MC_SetPosition_J5.Execute:=TRUE;
_MC_SetPosition_J6.Execute:=TRUE;
END_METHOD

METHOD M_StartHoming : BOOL
IF _SequenceMain = STEP_IDLE THEN
	M_StartHoming := TRUE;
	_StartHoming := TRUE;
ELSE
	M_StartHoming := FALSE;
END_IF
END_METHOD

END_FUNCTION_BLOCK

// ---- FB/move/MoveCmdProcessor.TcPOU
FUNCTION_BLOCK MoveCmdProcessor EXTENDS Module
VAR_INPUT
	Velocity: LREAL:=1000.0;
	VelFactor: LREAL:=1.0;
	Acceleration: LREAL:=1000.0;
	AccFactor: LREAL:=0.5;
	Jerk: LREAL:=1000.0;
	JerkFactor: LREAL:=0.5;
	Command: STRING(GVL.COMMAND_LEN):='';
END_VAR
VAR_IN_OUT
	AxisGroup: AXES_GROUP_REF;
	GroupHandler: FB_GroupHandler;
END_VAR
VAR_OUTPUT
	Position: DUT_COORD_REF;
END_VAR
VAR
	_SequenceSetCoordTrans: INT;
	_SequenceMoveCircularAbsolute: INT;
	_SequenceMoveCircularRelative: INT;
	_SequenceMoveDirectAbsolute: INT;
	_SequenceMoveDirectRelative: INT;
	_SequenceMoveLinearAbsolute: INT;
	_SequenceMoveLinearRelative: INT;
	_MC_GroupHalt: MC_GroupHalt;
	
	_MC_SetCoordinateTransformPreparation: MC_SetCoordinateTransformPreparation;
	_MC_MoveCircularAbsolutePreparation: MC_MoveCircularAbsolutePreparation;
	_MC_MoveLinearAbsolutePreparation: MC_MoveLinearAbsolutePreparation;
	
	_CoordRef: MC_COORD_REF;
	_buffer: ARRAY[1..4096] OF BYTE;
	_path: MC_PATH_DATA_REF(ADR(_buffer), SIZEOF(_buffer));
    _TargetPos: ARRAY[1.._NumberOfAxes] OF MC_LREAL;
    _TargetPos2: ARRAY[1.._NumberOfAxes] OF MC_LREAL;
    _TransitionParam: ARRAY[1..2] OF MC_LREAL;
    _MovePrepError: BOOL;
    _MC_MovePath: MC_MovePath;
	
	_UnitModeCurrentState: PACK_ML.State;
	_MoveCommandParser: ParseMoveCmd;
	_PosRef: DUT_COORD_REF;
	_PosRef2: DUT_COORD_REF;
	
	_MC_MoveRelative: ARRAY[1.._NumberOfAxes] OF MC_MoveRelative;
	_MoveDistance: ARRAY[1.._NumberOfAxes] OF LREAL:=[0,0,0,0,0,0];
	_MC_MoveAbsolute: ARRAY[1.._NumberOfAxes] OF MC_MoveAbsolute;
	_MovePosition: ARRAY[1.._NumberOfAxes] OF LREAL:=[0,0,0,0,0,0];
	
	_i, _j, _k: UINT;
END_VAR
VAR CONSTANT
	_NumberOfAxes:				UINT := GVL.NumberOfAxes;
	_STEP_DONE: 				INT := 1000;
	_STEP_IDLE: 				INT := 0000;
	_STEP_COMMAND: 				INT := 0020;
	_STEP_GROUP_POWER_ON: 		INT := 0022;
	_STEP_WAIT_POWER_ON: 		INT := 0024;
	_STEP_GROUP_ENABLE: 		INT := 0030;
	_STEP_WAIT_ENABLE: 			INT := 0035;
	_STEP_READ_POSITION: 		INT := 0040;
	_STEP_WAIT_POSITION: 		INT := 0050;
	_STEP_SET_KINEMATICS: 		INT := 0060;
	_STEP_WAIT_KINEMATICS: 		INT := 0070;
	_STEP_SET_COORD_TRANS:		INT := 0071;
	_STEP_WAIT_COORD_TRANS:		INT := 0072;
	_STEP_MOVE_TYPE:			INT := 0080;
	_STEP_WAIT_MOVE: 			INT := 0090;
	_STEP_GROUP_DISABLE: 		INT := 0100;
	_STEP_WAIT_DISABLE: 		INT := 0110;
	_STEP_GROUP_POWER_OFF: 		INT := 0120;
	_STEP_ERR: 					INT := 9999;
END_VAR

SUPER^();

// PackML state machine implementation
_UnitModeCurrentState := SUPER^._UnitMode.CurrentState;

//
CASE SUPER^._SeqMain OF
	
	_STEP_DONE:
		SUPER^._SeqMain := _STEP_IDLE;
		
	_STEP_IDLE:
		// wait here until commanded to start
		
	_STEP_COMMAND: // parse command
		_MoveCommandParser(Command:=Command);
		SUPER^._SeqMain := _STEP_GROUP_ENABLE;
		
	_STEP_GROUP_ENABLE:
		IF GroupHandler.M_EnableGroup(_MoveCommandParser.stCommand.CoordSystem) THEN
			SUPER^._SeqMain := _STEP_WAIT_ENABLE;
		ELSE
			(*SUPER^.M_Error(Description:=CONCAT('Group Handler Error: ',
										CONCAT(TO_STRING(GroupHandler.ErrorID),
										CONCAT(' ', SMC_ErrorString(GroupHandler.ErrorID,
													SMC_Language_Type.english)))));*)
			SUPER^.M_Error(Description:=CONCAT('Group Handler Error: ', TO_STRING(GroupHandler.ErrorID)));
			SUPER^._SeqMain := _STEP_ERR; // error step so we dont spam errors
		END_IF
		
	_STEP_WAIT_ENABLE:
		// TODO add timeout timer here?
		IF GroupHandler.P_GroupReady THEN
			SUPER^._SeqMain := _STEP_MOVE_TYPE;
		END_IF;
		
	_STEP_MOVE_TYPE: // parse move type
		_PosRef := _MoveCommandParser.stCommand.CoordRef;
		_PosRef2 := _MoveCommandParser.stCommand.CoordRef2; // the second position here is used for circular moves
		
		IF _MoveCommandParser.stCommand.MoveType = DUT_Command_MoveType.CircularMove THEN
			IF _MoveCommandParser.stCommand.PositionType = DUT_Command_PositionType.AbsolutePosition THEN
				_SequenceMoveCircularAbsolute := 1;
			ELSIF _MoveCommandParser.stCommand.PositionType = DUT_Command_PositionType.RelativePosition THEN
				_SequenceMoveCircularRelative := 1;
			END_IF
			
		ELSIF _MoveCommandParser.stCommand.MoveType = DUT_Command_MoveType.DirectMove THEN
			IF _MoveCommandParser.stCommand.PositionType = DUT_Command_PositionType.AbsolutePosition THEN
				_SequenceMoveDirectAbsolute := 1;
			ELSIF _MoveCommandParser.stCommand.PositionType = DUT_Command_PositionType.RelativePosition THEN
				_SequenceMoveDirectRelative := 1;
			END_IF
			
		ELSIF _MoveCommandParser.stCommand.MoveType = DUT_Command_MoveType.LinearMove THEN
			IF _MoveCommandParser.stCommand.PositionType = DUT_Command_PositionType.AbsolutePosition THEN
				_SequenceMoveLinearAbsolute := 1;
			ELSIF _MoveCommandParser.stCommand.PositionType = DUT_Command_PositionType.RelativePosition THEN
				_SequenceMoveLinearRelative := 1;
			END_IF
		END_IF
		
		SUPER^._SeqMain := _STEP_WAIT_MOVE;
		
	_STEP_WAIT_MOVE: // wait for move complete
		IF _SequenceMoveCircularAbsolute = 0
			AND _SequenceMoveCircularRelative = 0 
			AND _SequenceMoveDirectAbsolute = 0 
			AND _SequenceMoveDirectRelative = 0
			AND _SequenceMoveLinearAbsolute = 0
			AND _SequenceMoveLinearRelative = 0 THEN
				SUPER^._SeqMain := _STEP_GROUP_DISABLE;
				//SUPER^._SeqMain := _STEP_DONE;
		END_IF
	
	// TODO do we need to disable the group at this point? lets leave this here for now but skip it.
	_STEP_GROUP_DISABLE: 
		IF GroupHandler.M_DisableGroup() THEN
			SUPER^._SeqMain := _STEP_WAIT_DISABLE;
		ELSE
			(*SUPER^.M_Error(Description:=CONCAT('Group Handler Error: ',
										CONCAT(TO_STRING(GroupHandler.ErrorID),
										CONCAT(' ', SMC_ErrorString(GroupHandler.ErrorID,
													SMC_Language_Type.english)))));*)
			SUPER^.M_Error(Description:=CONCAT('Group Handler Error: ', TO_STRING(GroupHandler.ErrorID)));
			SUPER^._SeqMain := _STEP_ERR; // error step so we dont spam errors
		END_IF
		
	_STEP_WAIT_DISABLE:
		IF NOT GroupHandler.P_GroupReady THEN
			SUPER^._SeqMain := _STEP_DONE;
		END_IF
	
END_CASE

CASE _SequenceMoveCircularAbsolute OF
	0: //
	
	1: //
		_MC_MovePath.Execute := FALSE;
		A_AddLinAbsCircPath();
		_SequenceMoveCircularAbsolute := _SequenceMoveCircularAbsolute + 1;
		
	2: // 
		// TODO add timeout timer here
		IF _MovePrepError THEN
			(*SUPER^.M_Error(Description:=CONCAT('Move Command Error: ',
										CONCAT(TO_STRING(_MC_MoveLinearAbsolute.ErrorID),
										CONCAT(' ', SMC_ErrorString(_MC_MoveLinearAbsolute.ErrorID,
													SMC_Language_Type.english)))));*)
			//SUPER^.M_Error(Description:=CONCAT('Move Command Error: ', TO_STRING(_MC_MoveLinearAbsolute.ErrorID)));
			_SequenceMoveCircularAbsolute := 99; // error step so we dont spam errors
			
		ELSE
			_SequenceMoveCircularAbsolute := _SequenceMoveCircularAbsolute + 1;
		END_IF
		
	3: //
		_MC_MovePath.Execute := TRUE;
		_SequenceMoveCircularAbsolute := _SequenceMoveCircularAbsolute + 1;
		
	4: //
		// TODO add timeout timer here
		IF _MC_MovePath.Error THEN
			(*SUPER^.M_Error(Description:=CONCAT('Move Command Error: ',
										CONCAT(TO_STRING(_MC_MoveLinearAbsolute.ErrorID),
										CONCAT(' ', SMC_ErrorString(_MC_MoveLinearAbsolute.ErrorID,
													SMC_Language_Type.english)))));*)
			SUPER^.M_Error(Description:=CONCAT('Move Command Error: ', TO_STRING(_MC_MovePath.ErrorID)));
			_SequenceMoveCircularAbsolute := 99; // error step so we dont spam errors
			
		ELSIF _MC_MovePath.Done THEN
			_SequenceMoveCircularAbsolute := 0;
			
		END_IF
		
END_CASE

// CASE _SequenceMoveCircularRelative OF
// 	0: //
// 	
// 	1: //
// 		_MC_MoveCircularRelative.Execute := TRUE;
// 		_SequenceMoveCircularRelative := 2;
// 		
// 	2: //
// 		IF _MC_MoveCircularRelative.Error THEN
// 			(*SUPER^.M_Error(Description:=CONCAT('Move Command Error: ',
// 										CONCAT(TO_STRING(_MC_MoveCircularRelative.ErrorID),
// 										CONCAT(' ', SMC_ErrorString(_MC_MoveCircularRelative.ErrorID,
// 													SMC_Language_Type.english)))));*)
// 			SUPER^.M_Error(Description:=CONCAT('Move Command Error: ', TO_STRING(_MC_MoveCircularRelative.ErrorID)));
// 			_SequenceMoveCircularRelative := 3; // error step so we dont spam errors
// 		ELSIF  _MC_MoveCircularRelative.Done THEN
// 			_MC_MoveCircularRelative.Execute := FALSE;
// 			_SequenceMoveCircularRelative := 0;
// 		END_IF
// 		
// END_CASE

// CASE _SequenceMoveDirectAbsolute OF
// 	0: //
// 	
// 	1: //
// 		_MC_MoveDirectAbsolute.Execute := TRUE;
// 		_SequenceMoveDirectAbsolute := 2;
// 		
// 	2: //
// 		IF _MC_MoveDirectAbsolute.Error THEN
// 			(*SUPER^.M_Error(Description:=CONCAT('Move Command Error: ',
// 										CONCAT(TO_STRING(_MC_MoveDirectAbsolute.ErrorID),
// 										CONCAT(' ', SMC_ErrorString(_MC_MoveDirectAbsolute.ErrorID,
// 													SMC_Language_Type.english)))));*)
// 			SUPER^.M_Error(Description:=CONCAT('Move Command Error: ', TO_STRING(_MC_MoveDirectAbsolute.ErrorID)));
// 			_SequenceMoveDirectAbsolute := 3; // error step so we dont spam errors
// 			
// 		ELSIF _MC_MoveDirectAbsolute.Done THEN
// 			_MC_MoveDirectAbsolute.Execute := FALSE;
// 			_SequenceMoveDirectAbsolute := 0;
// 		END_IF
// 		
// END_CASE

// CASE _SequenceMoveDirectRelative OF
// 	0: //
// 	
// 	1: //
// 		_MC_MoveDirectRelative.Execute := TRUE;
// 		_SequenceMoveDirectRelative := 2;
// 		
// 	2: //
// 		IF _MC_MoveDirectRelative.Error THEN
// 			(*SUPER^.M_Error(Description:=CONCAT('Move Command Error: ',
// 										CONCAT(TO_STRING(_MC_MoveDirectRelative.ErrorID),
// 										CONCAT(' ', SMC_ErrorString(_MC_MoveDirectRelative.ErrorID,
// 													SMC_Language_Type.english)))));*)
// 			SUPER^.M_Error(Description:=CONCAT('Move Command Error: ', TO_STRING(_MC_MoveDirectRelative.ErrorID)));
// 			_SequenceMoveDirectRelative := 3; // error step so we dont spam errors
// 			
// 		ELSIF _MC_MoveDirectRelative.Done THEN
// 			_MC_MoveDirectRelative.Execute := FALSE;
// 			_SequenceMoveDirectRelative := 0;
// 		END_IF
// 		
// END_CASE

CASE _SequenceMoveLinearAbsolute OF
	0: //
	
	1: //
		_MC_MovePath.Execute := FALSE;
		A_AddLinAbsPath();
		_SequenceMoveLinearAbsolute := _SequenceMoveLinearAbsolute + 1;
		
	2: // 
		// TODO add timeout timer here
		IF _MovePrepError THEN
			(*SUPER^.M_Error(Description:=CONCAT('Move Command Error: ',
										CONCAT(TO_STRING(_MC_MoveLinearAbsolute.ErrorID),
										CONCAT(' ', SMC_ErrorString(_MC_MoveLinearAbsolute.ErrorID,
													SMC_Language_Type.english)))));*)
			//SUPER^.M_Error(Description:=CONCAT('Move Command Error: ', TO_STRING(_MC_MoveLinearAbsolute.ErrorID)));
			_SequenceMoveLinearAbsolute := 99; // error step so we dont spam errors
			
		ELSE
			_SequenceMoveLinearAbsolute := _SequenceMoveLinearAbsolute + 1;
		END_IF
		
	3: //
		_MC_MovePath.Execute := TRUE;
		_SequenceMoveLinearAbsolute := _SequenceMoveLinearAbsolute + 1;
		
	4: //
		// TODO add timeout timer here
		IF _MC_MovePath.Error THEN
			(*SUPER^.M_Error(Description:=CONCAT('Move Command Error: ',
										CONCAT(TO_STRING(_MC_MoveLinearAbsolute.ErrorID),
										CONCAT(' ', SMC_ErrorString(_MC_MoveLinearAbsolute.ErrorID,
													SMC_Language_Type.english)))));*)
			SUPER^.M_Error(Description:=CONCAT('Move Command Error: ', TO_STRING(_MC_MovePath.ErrorID)));
			_SequenceMoveLinearAbsolute := 99; // error step so we dont spam errors
			
		ELSIF _MC_MovePath.Done THEN
			_SequenceMoveLinearAbsolute := 0;
			
		END_IF
		
END_CASE

// CASE _SequenceMoveLinearRelative OF
// 	0: //
// 	
// 	1: //
// 		_MC_MoveLinearRelative.Execute := TRUE;
// 		_SequenceMoveLinearRelative := 2;
// 		
// 	2: //
// 		IF _MC_MoveLinearRelative.Error THEN
// 		    (*SUPER^.M_Error(Description:=CONCAT('Move Command Error: ',
// 										CONCAT(TO_STRING(_MC_MoveLinearRelative.ErrorID),
// 										CONCAT(' ', SMC_ErrorString(_MC_MoveLinearRelative.ErrorID,
// 													SMC_Language_Type.english)))));*)
// 			SUPER^.M_Error(Description:=CONCAT('Move Command Error: ', TO_STRING(_MC_MoveLinearRelative.ErrorID)));
// 			_SequenceMoveLinearRelative := 3; // error step so we dont spam errors
// 			
// 		ELSIF _MC_MoveLinearRelative.Done THEN
// 			_MC_MoveLinearRelative.Execute := FALSE;
// 			_SequenceMoveLinearRelative := 0;
// 		END_IF
// 		
// END_CASE

_MC_GroupHalt(
	AxesGroup:= AxisGroup, 
	Execute:= , 
	Deceleration:= Acceleration, 
	Jerk:= JerkFactor, 
	Done=> , 
	Busy=> , 
	Active=> , 
	CommandAborted=> , 
	Error=> , 
	ErrorId=> );
	
_MC_MovePath(
	AxesGroup:= AxisGroup, 
	PathData:= _Path, 
	Execute:= , 
	Done=> , 
	Busy=> , 
	Active=> , 
	CommandAborted=> , 
	Error=> , 
	ErrorId=> );

// https://content.helpme-codesys.com/de/libs/SM3_Robotics/Current/SM3_Robotics/POUs/Movement/MC_MoveCircularAbsolute.html
// https://content.helpme-codesys.com/de/libs/SM3_Robotics/Current/SM3_Robotics/Basic-types/SMC_CIRC_MODE.html#smc-circ-mode
// _MC_MoveCircularAbsolute(
// 	AxisGroup:= AxisGroup, 
// 	Execute:= , 
// 	CircMode:= _MoveCommandParser.stCommand.CircleMode, 
// 	AuxPoint:= _PosRef, 
// 	EndPoint:= _PosRef2, 
// 	PathChoice:= _MoveCommandParser.stCommand.PathChoice, 
// 	Velocity:= Velocity, 
// 	Acceleration:= Acceleration, 
// 	Deceleration:= Acceleration, 
// 	Jerk:= Jerk, 
// 	CoordSystem:= _MoveCommandParser.stCommand.CoordSystem, 
// 	BufferMode:= , 
// 	TransitionMode:= , 
// 	TransitionParameter:= , 
// 	OrientationMode:= , 
// 	VelFactor:= SEL(_MoveCommandParser.stCommand.Speed > 100, _MoveCommandParser.stCommand.Speed / 100.0, 1), // cannot be greater than 1
// 	AccFactor:= SEL(AccFactor > 1, AccFactor, 1), 
// 	JerkFactor:= SEL(JerkFactor > 1, JerkFactor, 1), 
// 	TorqueFactor:= 1, 
// 	Done=> , 
// 	Busy=> , 
// 	Active=> , 
// 	CommandAborted=> , 
// 	CommandAccepted=> , 
// 	Error=> , 
// 	ErrorID=> , 
// 	MovementId=> );

// https://content.helpme-codesys.com/en/libs/SM3_Robotics/Current/SM3_Robotics/POUs/Movement/MC_MoveCircularRelative.html
// https://content.helpme-codesys.com/de/libs/SM3_Robotics/Current/SM3_Robotics/Basic-types/SMC_CIRC_MODE.html#smc-circ-mode
// _MC_MoveCircularRelative(
// 	AxisGroup:= AxisGroup, 
// 	Execute:= , 
// 	CircMode:= _MoveCommandParser.stCommand.CircleMode, 
// 	AuxPoint:= _PosRef, 
// 	EndPoint:= _PosRef2, 
// 	PathChoice:= _MoveCommandParser.stCommand.PathChoice, 
// 	Velocity:= Velocity, 
// 	Acceleration:= Acceleration, 
// 	Deceleration:= Acceleration, 
// 	Jerk:= Jerk, 
// 	CoordSystem:= _MoveCommandParser.stCommand.CoordSystem, 
// 	BufferMode:= , 
// 	TransitionMode:= , 
// 	TransitionParameter:= , 
// 	OrientationMode:= , 
// 	VelFactor:= SEL(_MoveCommandParser.stCommand.Speed > 100, _MoveCommandParser.stCommand.Speed / 100.0, 1), // cannot be greater than 1
// 	AccFactor:= SEL(AccFactor > 1, AccFactor, 1), 
// 	JerkFactor:= SEL(JerkFactor > 1, JerkFactor, 1), 
// 	TorqueFactor:= 1, 
// 	Done=> , 
// 	Busy=> , 
// 	Active=> , 
// 	CommandAborted=> , 
// 	CommandAccepted=> , 
// 	Error=> , 
// 	ErrorID=> , 
// 	MovementId=> );


// // move relative
// FOR _k:= 1 TO _NumberOfAxes DO
// 	_MC_MoveRelative[_k](
// 		Axis:= SEL(_MoveCommandParser.stCommand.CoordSystem = DUT_CoordSystem.ACS, MCS[_k], ACS[_k]), 
// 		Execute:= , 
// 		Distance:= _MoveDistance[_k], 
// 		Velocity:= _MoveCommandParser.stCommand.Speed, 
// 		Acceleration:= MC_DEFAULT, 
// 		Deceleration:= MC_DEFAULT, 
// 		Jerk:= MC_DEFAULT, 
// 		BufferMode:= , 
// 		Options:= , 
// 		Done=> , 
// 		Busy=> , 
// 		Active=> , 
// 		CommandAborted=> , 
// 		Error=> , 
// 		ErrorID=> );
// END_FOR

// FOR _k:= 1 TO _NumberOfAxes DO
// 	_MC_MoveAbsolute[_k](
// 		Axis:= SEL(_MoveCommandParser.stCommand.CoordSystem = DUT_CoordSystem.ACS, MCS[_k], ACS[_k]), 
// 		Execute:= , 
// 		Position:= _MovePosition[_k], 
// 		Velocity:= _MoveCommandParser.stCommand.Speed, 
// 		Acceleration:= MC_DEFAULT, 
// 		Deceleration:= MC_DEFAULT, 
// 		Jerk:= MC_DEFAULT, 
// 		BufferMode:= , 
// 		Options:= , 
// 		Done=> , 
// 		Busy=> , 
// 		Active=> , 
// 		CommandAborted=> , 
// 		Error=> , 
// 		ErrorID=> );
// END_FOR

// _MC_MoveDirectAbsolute(
// 	AxisGroup:=AxisGroup,
// 	Execute:= ,
// 	Position:= _PosRef,
// 	MovementType:= ,
// 	CoordSystem:= _MoveCommandParser.stCommand.CoordSystem,
// 	BufferMode:= ,
// 	TransitionMode:= ,
// 	TransitionParameter:= ,
// 	VelFactor:= SEL(_MoveCommandParser.stCommand.Speed > 100, _MoveCommandParser.stCommand.Speed / 100.0, 1), // cannot be greater than 1
// 	AccFactor:= SEL(AccFactor > 1, AccFactor, 1), 
// 	JerkFactor:= SEL(JerkFactor > 1, JerkFactor, 1), 
// 	TorqueFactor:= 1,
// 	Done=> ,
// 	Busy=> ,
// 	Active=> ,
// 	CommandAborted=> ,
// 	CommandAccepted=> ,
// 	Error=> ,
// 	ErrorID=> ,
// 	MovementId=> );

// _MC_MoveDirectRelative(
// 	AxisGroup:= AxisGroup, 
// 	Execute:= , 
// 	Distance:= _PosRef, 
// 	MovementType:= , 
// 	CoordSystem:= _MoveCommandParser.stCommand.CoordSystem, 
// 	BufferMode:= , 
// 	TransitionMode:= , 
// 	TransitionParameter:= , 
// 	VelFactor:= SEL(_MoveCommandParser.stCommand.Speed > 100, _MoveCommandParser.stCommand.Speed / 100.0, 1), // cannot be greater than 1
// 	AccFactor:= SEL(AccFactor > 1, AccFactor, 1), 
// 	JerkFactor:= SEL(JerkFactor > 1, JerkFactor, 1), 
// 	TorqueFactor:= 1, 
// 	Done=> , 
// 	Busy=> , 
// 	Active=> , 
// 	CommandAborted=> , 
// 	CommandAccepted=> , 
// 	Error=> , 
// 	ErrorID=> , 
// 	MovementId=> );
	
// _MC_MoveLinearAbsolute(
// 	AxisGroup:= AxisGroup, 
// 	Execute:= , 
// 	Position:= _PosRef,
// 	Velocity:= 1000, 
// 	Acceleration:= Acceleration, 
// 	Deceleration:= Acceleration, 
// 	Jerk:= Jerk, 
// 	CoordSystem:= _MoveCommandParser.stCommand.CoordSystem, 
// 	BufferMode:= , 
// 	TransitionMode:= , 
// 	TransitionParameter:= , 
// 	OrientationMode:= , 
// 	VelFactor:= SEL(_MoveCommandParser.stCommand.Speed > 100, _MoveCommandParser.stCommand.Speed / 100.0, 1), // cannot be greater than 1
// 	AccFactor:= SEL(AccFactor > 1, AccFactor, 1), 
// 	JerkFactor:= SEL(JerkFactor > 1, JerkFactor, 1), 
// 	TorqueFactor:= 1, 
// 	Done=> , 
// 	Busy=> , 
// 	Active=> , 
// 	CommandAborted=> , 
// 	CommandAccepted=> , 
// 	Error=> , 
// 	ErrorID=> , 
// 	MovementId=> );
	
// _MC_MoveLinearRelative(
// 	AxisGroup:= AxisGroup, 
// 	Execute:= , 
// 	Distance:= _PosRef, 
// 	Velocity:= 1000, 
// 	Acceleration:= Acceleration, 
// 	Deceleration:= Acceleration, 
// 	Jerk:= Jerk, 
// 	CoordSystem:= _MoveCommandParser.stCommand.CoordSystem, 
// 	BufferMode:= , 
// 	TransitionMode:= , 
// 	TransitionParameter:= , 
// 	OrientationMode:= , 
// 	VelFactor:= SEL(_MoveCommandParser.stCommand.Speed > 100, _MoveCommandParser.stCommand.Speed / 100.0, 1), // cannot be greater than 1
// 	AccFactor:= SEL(AccFactor > 1, AccFactor, 1), 
// 	JerkFactor:= SEL(JerkFactor > 1, JerkFactor, 1), 
// 	TorqueFactor:= 1, 
// 	Done=> , 
// 	Busy=> , 
// 	Active=> , 
// 	CommandAborted=> , 
// 	CommandAccepted=> , 
// 	Error=> , 
// 	ErrorID=> , 
// 	MovementId=> );

ACTION A_AddLinAbsCircPath:
_MovePrepError := FALSE;
_path.ClearPath();  //Clear nodes that were in path

//
CASE _MoveCommandParser.stCommand.CoordSystem OF
	DUT_CoordSystem.ACS:
		_CoordRef := GVL.McsCoordRef; // TODO: we shouldnt be here. maybe fault?
	DUT_CoordSystem.MCS:
		_CoordRef := GVL.McsCoordRef;
	DUT_CoordSystem.UCS1:
		_CoordRef := GVL.Ucs1CoordRef;
	DUT_CoordSystem.UCS2:
		_CoordRef := GVL.Ucs2CoordRef;
	DUT_CoordSystem.TCP:
		_CoordRef := GVL.TcpCoordRef;
END_CASE
_MC_SetCoordinateTransformPreparation(PathData:=_path, CoordTransform:=_CoordRef);
_MovePrepError := _MovePrepError OR _MC_SetCoordinateTransformPreparation.Error;

_TargetPos[1]				:= _PosRef.X;
_TargetPos[2]				:= _PosRef.Y;
_TargetPos[3]				:= _PosRef.Z;
_TargetPos[4]				:= GroupHandler.P_GroupStatus.CurrentPosition.A + _PosRef.A;
_TargetPos[5]				:= GroupHandler.P_GroupStatus.CurrentPosition.B + _PosRef.B;
_TargetPos[6]				:= GroupHandler.P_GroupStatus.CurrentPosition.C + _PosRef.C;
_TargetPos2[1]				:= _PosRef2.X;
_TargetPos2[2]				:= _PosRef2.Y;
_TargetPos2[3]				:= _PosRef2.Z;
_TargetPos2[4]				:= GroupHandler.P_GroupStatus.CurrentPosition.A + _PosRef.A;
_TargetPos2[5]				:= GroupHandler.P_GroupStatus.CurrentPosition.B + _PosRef.B;
_TargetPos2[6]				:= GroupHandler.P_GroupStatus.CurrentPosition.C + _PosRef.C;
_TransitionParam[1]			:= 0; //blending distance on previous segment, no influence here
_TransitionParam[2]			:= 0; //blending distance on this segment, no influence here

_MC_MoveCircularAbsolutePreparation(
	PathData:= _path, 
	CircMode:= _MoveCommandParser.stCommand.CircleMode, 
	AuxPoint:= ADR(_TargetPos), 
	AuxPointCount:= 3, 
	EndPoint:= ADR(_TargetPos2), 
	EndPointCount:= _NumberOfAxes, 
	PathChoice:= _MoveCommandParser.stCommand.PathChoice, 
	Velocity:= _MoveCommandParser.stCommand.Speed, 
	Acceleration:= MC_DEFAULT, 
	Deceleration:= MC_DEFAULT, 
	Jerk:= MC_DEFAULT, 
	BufferMode:= mcBlendingPrevious, 
	TransitionMode:= mcTransModeCornerDistanceAdvanced, 
	TransitionParameter:= ADR (_TransitionParam), 
	TransitionParameterCount:= 2, 
	InvokeId:= 10, // TODO should increment this with each additional call made here if calls are added
	DynamicConstraints:= , 
	Error=> , 
	ErrorId=> );
_MovePrepError := _MovePrepError OR _MC_MoveCircularAbsolutePreparation.Error;
END_ACTION

ACTION A_AddLinAbsPath:
_MovePrepError := FALSE;
_path.ClearPath();  //Clear nodes that were in path

_MC_MoveLinearAbsolutePreparation.Position						:= ADR(_TargetPos); //pointer to position array
_MC_MoveLinearAbsolutePreparation.PositionCount 				:= _NumberOfAxes; //number of axes in group
_MC_MoveLinearAbsolutePreparation.TransitionParameter			:= ADR (_TransitionParam); //pointer to transition parameter array
_MC_MoveLinearAbsolutePreparation.TransitionParameterCount		:= 2; //number of transition parameters, has to be set always 2
_MC_MoveLinearAbsolutePreparation.BufferMode					:= mcBlendingPrevious;
_MC_MoveLinearAbsolutePreparation.TransitionMode				:= mcTransModeCornerDistanceAdvanced;
//Set dynamics to default values of the axes
_MC_MoveLinearAbsolutePreparation.Acceleration					:= MC_DEFAULT;
_MC_MoveLinearAbsolutePreparation.Deceleration					:= MC_DEFAULT;
_MC_MoveLinearAbsolutePreparation.Jerk							:= MC_DEFAULT;

//
CASE _MoveCommandParser.stCommand.CoordSystem OF
	DUT_CoordSystem.ACS:
		_CoordRef := GVL.McsCoordRef; // TODO: we shouldnt be here. maybe fault?
	DUT_CoordSystem.MCS:
		_CoordRef := GVL.McsCoordRef;
	DUT_CoordSystem.UCS1:
		_CoordRef := GVL.Ucs1CoordRef;
	DUT_CoordSystem.UCS2:
		_CoordRef := GVL.Ucs2CoordRef;
	DUT_CoordSystem.TCP:
		_CoordRef := GVL.TcpCoordRef;
END_CASE
_MC_SetCoordinateTransformPreparation(PathData:=_path, CoordTransform:=_CoordRef);
_MovePrepError := _MovePrepError OR _MC_SetCoordinateTransformPreparation.Error;

//1st node
_TargetPos[1]				:= _PosRef.X;
_TargetPos[2]				:= _PosRef.Y;
_TargetPos[3]				:= _PosRef.Z;
// _TargetPos[4]				:= GroupHandler.P_GroupStatus.CurrentPosition.A + _PosRef.A;
// _TargetPos[5]				:= GroupHandler.P_GroupStatus.CurrentPosition.B + _PosRef.B;
// _TargetPos[6]				:= GroupHandler.P_GroupStatus.CurrentPosition.C + _PosRef.C;
_TargetPos[4]				:= _PosRef.A;
_TargetPos[5]				:= _PosRef.B;
_TargetPos[6]				:= _PosRef.C;
_TransitionParam[1]			:= 0; //blending distance on previous segment, no influence here
_TransitionParam[2]			:= 0; //blending distance on this segment, no influence here
_MC_MoveLinearAbsolutePreparation(	PathData:= _path,
									Velocity:= _MoveCommandParser.stCommand.Speed, 
									InvokeId:= 10); // TODO should increment this with each additional call made here if calls are added
_MovePrepError := _MovePrepError OR _MC_MoveLinearAbsolutePreparation.Error;
END_ACTION

ACTION A_AddLinRelPath:

END_ACTION

METHOD PROTECTED M_Aborting : BOOL
CASE _SeqAborting OF
	0:
		GroupHandler.M_DisableGroup();
		_SeqAborting := _SeqAborting + 1;
	1:
		IF NOT GroupHandler.P_GroupReady THEN
			SUPER^.M_StateComplete();
			_SeqAborting := 0;
		END_IF
		
END_CASE
END_METHOD

METHOD PROTECTED M_Clearing : BOOL

_MC_MovePath.Execute := FALSE;
_SequenceMoveCircularAbsolute := 0;
_SequenceMoveCircularRelative := 0;
_SequenceMoveDirectAbsolute := 0;
_SequenceMoveDirectRelative := 0;
_SequenceMoveLinearAbsolute := 0;
_SequenceMoveLinearRelative := 0;
_SequenceSetCoordTrans := 0;

SUPER^.M_StateComplete();
END_METHOD

METHOD PROTECTED M_Complete : BOOL
// once complete, reset to get back to idle
SUPER^._UnitMode.Reset();
END_METHOD

METHOD PROTECTED M_Execute : BOOL
// here we want to execute our commands/jobs/etc and set completed when done.
IF SUPER^._SeqMain =_STEP_IDLE THEN
	SUPER^.M_StateComplete();
END_IF
END_METHOD

METHOD PROTECTED M_Holding : BOOL
CASE SUPER^._SeqHolding OF
	0:
		_MC_MovePath.Execute := FALSE;
		_MC_GroupHalt.Execute:=TRUE;
		_SeqHolding := _SeqHolding + 1;
	1:
		IF _MC_GroupHalt.Done THEN
			_MC_GroupHalt.Execute := FALSE;
			SUPER^.M_StateComplete();
			_SeqHolding := 0;
		END_IF
		
END_CASE
END_METHOD

METHOD PROTECTED M_Idle : BOOL
// in this state, we want to reset all the function blocks and hang out

_MC_MovePath.Execute := FALSE;
_SequenceMoveCircularAbsolute := 0;
_SequenceMoveCircularRelative := 0;
_SequenceMoveDirectAbsolute := 0;
_SequenceMoveDirectRelative := 0;
_SequenceMoveLinearAbsolute := 0;
_SequenceMoveLinearRelative := 0;
_SequenceSetCoordTrans := 0;
SUPER^._SeqMain := 0;
END_METHOD

METHOD PROTECTED M_Resetting : BOOL
CASE SUPER^._SeqResetting OF
	0:
		GroupHandler.M_ResetGroup();
		SUPER^._SeqResetting := SUPER^._SeqResetting + 1;
	1:
		// needed to add this here as a hack to make sure keep in lock step with the reset sequence.
		// i think ideally, i should add a "is reset" property.
		IF GroupHandler.Busy THEN
			SUPER^._SeqResetting := SUPER^._SeqResetting + 1;
		END_IF
	2:
		IF NOT GroupHandler.Busy THEN
			SUPER^.M_StateComplete();
			SUPER^._SeqResetting := 0;
		END_IF
END_CASE
END_METHOD

METHOD PROTECTED M_SetPackML : BOOL
SUPER^._UnitMode(	sName := 'Move Processor',
				eInitialState := PACK_ML.State.Idle,
				xActive := TRUE);
END_METHOD

METHOD PROTECTED M_Starting : BOOL
// here we want to clear things and get ready for the execute state
// I can consider this the "INIT" state
SUPER^._SeqMain := _STEP_COMMAND;
SUPER^.M_StateComplete();
END_METHOD

METHOD PROTECTED M_UnHolding : BOOL
// here the operator called unhold (most likely from M_Start)
_MC_GroupHalt.Execute := FALSE;
_MC_MovePath.Execute := TRUE;
CASE _MoveCommandParser.stCommand.MoveType OF 
	DUT_Command_MoveType.DirectMove:
		IF _MoveCommandParser.stCommand.PositionType = DUT_Command_Positiontype.AbsolutePosition THEN
			//_MC_MoveDirectAbsolute.Execute := TRUE;
		ELSE
			//_MC_MoveDirectRelative.Execute := TRUE;
		END_IF
	DUT_Command_MoveType.LinearMove:
		IF _MoveCommandParser.stCommand.PositionType = DUT_Command_Positiontype.AbsolutePosition THEN
			//_MC_MoveLinearAbsolute.Execute := TRUE;
		ELSE
			//_MC_MoveLinearRelative.Execute := TRUE;
		END_IF
	DUT_Command_MoveType.CircularMove:
		IF _MoveCommandParser.stCommand.PositionType = DUT_Command_Positiontype.AbsolutePosition THEN
			//_MC_MoveCircularAbsolute.Execute := TRUE;
		ELSE
			//_MC_MoveCircularRelative.Execute := TRUE;
		END_IF
END_CASE
//
SUPER^.M_StateComplete();
END_METHOD

END_FUNCTION_BLOCK

// ---- FB/template/Module.TcPOU
FUNCTION_BLOCK Module EXTENDS PackML IMPLEMENTS ItfModule

VAR_INPUT // input vars
	StoredPositions: REFERENCE TO ARRAY[GVL.POS_ARR_BEG..GVL.POS_ARR_END] OF DUT_StoredPosition;
	VisionRegisters: REFERENCE TO ARRAY[GVL.VIS_ARR_BEG..GVL.VIS_ARR_END] OF DUT_VisionRegister;
	Flags: REFERENCE TO ARRAY[GVL.FLG_ARR_BEG..GVL.FLG_ARR_END] OF DUT_Flags;
END_VAR

VAR_OUTPUT // output vars
	ItfUnitMode: PACK_ML.IUnitMode;
	Busy: BOOL;
	Error: BOOL;
	ErrorDescription: STRING;
END_VAR

VAR // standard local vars
	_TimeoutTimer: TON:=(PT:=T#0MS);
	_Home, _Start: BOOL;
	_ModuleFirstScan: BOOL:=TRUE;
	_SeqStart, _SeqHome: INT;
	_AbortedRtrig: R_Trig;
END_VAR

VAR CONSTANT //
	STEP_IDLE: INT := 0000;
	STEP_DONE: INT := 0020;
	STEP_RUN:  INT := 0030;
END_VAR

SUPER^();

//
IF _ModuleFirstScan THEN
	ItfUnitMode := SUPER^.IUnitMode;
END_IF;

//
_M_Home();
_M_Start();

//
Busy := _UnitMode.CurrentState <> PACK_ML.State.Idle
		AND _UnitMode.CurrentState <> PACK_ML.State.Aborted
		AND _UnitMode.CurrentState <> PACK_ML.State.Complete
		AND _UnitMode.CurrentState <> PACK_ML.State.Held
		AND _UnitMode.CurrentState <> PACK_ML.State.Stopped
		AND _UnitMode.CurrentState <> PACK_ML.State.Suspended;
		
//
_AbortedRtrig(CLK:=_UnitMode.CurrentState = PACK_ML.State.Aborted);
IF _AbortedRtrig.Q THEN
	//_SeqStart := 0;  _Start:=FALSE;
	//_SeqHome := 0; _Home:=FALSE;
END_IF

//
_TimeoutTimer(IN:= Busy AND _TimeoutTimer.PT > T#0MS); // ignore if timer set to 0
IF _TimeoutTimer.Q THEN
	M_Error(Description:= CONCAT('Task timed out after ', TIME_TO_STRING(_TimeoutTimer.ET)));
END_IF

// do not place anything below this
_ModuleFirstScan:=FALSE;

METHOD PRIVATE _M_Home : BOOL
CASE _SeqHome OF
	0:
		//
		IF _Home THEN
			_Home := FALSE;
			M_Reset();
			_SeqHome := _SeqHome + 1;
		END_IF
	1:
		//
		CASE _UnitMode.CurrentState OF
			PACK_ML.State.Aborted:
				_UnitMode.Clear();
				
			PACK_ML.State.Stopped,
			PACK_ML.State.Complete:
				_UnitMode.Reset();
				_SeqHome := _SeqHome + 1;
				
			PACK_ML.State.Resetting,
			PACK_ML.State.Clearing,
			PACK_ML.State.Aborting:
				// just wait
		ELSE
			_UnitMode.Abort();
			
		END_CASE
		
	2:
		IF _UnitMode.CurrentState = PACK_ML.State.Idle THEN
			_SeqHome := 0;
		END_IF
		
END_CASE
END_METHOD

METHOD PRIVATE _M_Start : BOOL
CASE _SeqStart OF
	0:
		IF _Start THEN
			_Start := FALSE;
			M_Reset();
			_SeqStart := _SeqStart + 1;
		END_IF
	1:
		CASE _UnitMode.CurrentState OF
			PACK_ML.State.Clearing,
			PACK_ML.State.Resetting,
			PACK_ML.State.UnHolding,
			PACK_ML.State.UnSuspending,
			PACK_ML.State.Starting:
				// be patient
			PACK_ML.State.Aborted:
				_UnitMode.Clear();
			PACK_ML.State.Stopped:
				_UnitMode.Reset();
			PACK_ML.State.Held:
				_UnitMode.UnHold();
			PACK_ML.State.Suspended:
				_UnitMode.UnSuspend();
			PACK_ML.State.Idle:
				_UnitMode.Start();
			PACK_ML.State.Execute:
				_SeqStart := 0;
		ELSE
			_SeqStart := 0;
		END_CASE
		
END_CASE
END_METHOD

METHOD M_Abort
_UnitMode.Abort();
_SeqStart := 0;  _Start:=FALSE;
_SeqHome := 0; _Home:=FALSE;
END_METHOD

METHOD PROTECTED M_Error : BOOL
VAR_INPUT
	Description: STRING;
END_VAR
// suspend state machine
_UnitMode.Suspend();

//
Error := TRUE;

//
IF ErrorDescription = '' THEN
	ErrorDescription := Description;
ELSE // add a space and tack on the additional error description
	ErrorDescription := CONCAT(ErrorDescription, ' ');
	ErrorDescription := CONCAT(ErrorDescription, Description);
END_IF
END_METHOD

METHOD M_Hold
_UnitMode.Hold();
END_METHOD

METHOD M_Home
_Home:=TRUE;
END_METHOD

METHOD PROTECTED M_Reset : BOOL
Error := FALSE;
ErrorDescription := '';
END_METHOD

METHOD M_Start
_Start := TRUE;
END_METHOD

METHOD M_Stop
_UnitMode.Stop();
END_METHOD

{attribute 'monitoring' := 'variable'}
PROPERTY PropBusy : BOOL
GET
PropBusy := Busy;
END_GET
END_PROPERTY

{attribute 'monitoring' := 'variable'}
PROPERTY PropCurrentState : PACK_ML.State
GET
PropCurrentState := ItfUnitMode.CurrentState;
END_GET
END_PROPERTY

{attribute 'monitoring' := 'variable'}
PROPERTY PropErrDescription : STRING
GET
PropErrDescription := ErrorDescription;
END_GET
END_PROPERTY

{attribute 'monitoring' := 'variable'}
PROPERTY PropError : BOOL
GET
PropError := Error;
END_GET
END_PROPERTY

END_FUNCTION_BLOCK

// ---- FB/template/PackML.TcPOU
{attribute 'reflection'}
FUNCTION_BLOCK PackML
VAR_INPUT
END_VAR
VAR_OUTPUT
	IUnitMode: PACK_ML.IUnitMode;
END_VAR
VAR
	 {attribute 'instance-path'}
	 {attribute 'noinit'}
	 instance_path: STRING(255);
	_UnitMode: PACK_ML.UnitMode;
	_StateTimer: TON;
	_PackMLFirstScan: BOOL:=TRUE;
	_SeqMain, _SeqAborting, _SeqClearing, _SeqCompleting, _SeqHolding, _SeqResetting,
	_SeqStarting, _SeqStopping, _SeqSuspending, _SeqUnholding, _SeqUnSuspending: INT;
END_VAR
VAR CONSTANT
	STATE_TIME: TIME := T#0MS;
END_VAR

//
IF _PackMLFirstScan THEN
	_PackMLFirstScan := FALSE;
	M_SetPackMl();
	IUnitMode := _UnitMode;
END_IF

//
_StateTimer(PT:=STATE_TIME);

//
CASE _UnitMode.CurrentState OF
	PACK_ML.State.Stopped:
		M_Stopped();
	PACK_ML.State.Aborted:
		M_Aborted();
	PACK_ML.State.Held:
		M_Held();
	PACK_ML.State.Suspended:
		M_Suspended();
	PACK_ML.State.Complete:
		M_Complete();
	PACK_ML.State.Idle:
		M_Idle();
	PACK_ML.State.Resetting:
		M_Resetting();
	PACK_ML.State.Starting:
		M_Starting();
	PACK_ML.State.Execute:
		M_Execute();
	PACK_ML.State.Suspending:
		M_Suspending();
	PACK_ML.State.UnSuspending:
		M_UnSuspending();
	PACK_ML.State.Holding:
		M_Holding();
	PACK_ML.State.UnHolding:
		M_UnHolding();
	PACK_ML.State.Completing:
		M_Completing();
	PACK_ML.State.Aborting:
		M_Aborting();
	PACK_ML.State.Stopping:
		M_Stopping();
	PACK_ML.State.Clearing:
		M_Clearing();
END_CASE

METHOD PROTECTED M_Aborted : BOOL
_SeqMain := 0;
_SeqAborting := 0;
_SeqClearing := 0;
_SeqCompleting := 0;
_SeqHolding := 0;
_SeqResetting := 0;
_SeqStarting := 0;
_SeqStopping := 0;
_SeqSuspending := 0;
_SeqUnholding := 0;
_SeqUnSuspending := 0;
END_METHOD

METHOD PROTECTED M_Aborting : BOOL
_StateTimer.IN:=TRUE;

IF _StateTimer.Q THEN
	_StateTimer.IN:=FALSE;
	M_StateComplete();
END_IF
END_METHOD

METHOD PROTECTED M_Clearing : BOOL
_StateTimer.IN:=TRUE;

IF _StateTimer.Q THEN
	_StateTimer.IN:=FALSE;
	M_StateComplete();
END_IF
END_METHOD

METHOD PROTECTED M_Complete : BOOL
(*_StateTimer.IN:=TRUE;

IF _StateTimer.Q THEN
	_StateTimer.IN:=FALSE;
	M_StateComplete();
END_IF*)
END_METHOD

METHOD PROTECTED M_Completing : BOOL
_StateTimer.IN:=TRUE;

IF _StateTimer.Q THEN
	_StateTimer.IN:=FALSE;
	M_StateComplete();
END_IF
END_METHOD

METHOD PROTECTED M_Execute : BOOL
END_METHOD

METHOD PROTECTED M_Held : BOOL
(*_StateTimer.IN:=TRUE;

IF _StateTimer.Q THEN
	_StateTimer.IN:=FALSE;
	M_StateComplete();
END_IF*)
END_METHOD

METHOD PROTECTED M_Holding : BOOL
_StateTimer.IN:=TRUE;

IF _StateTimer.Q THEN
	_StateTimer.IN:=FALSE;
	M_StateComplete();
END_IF
END_METHOD

METHOD PROTECTED M_Idle : BOOL
(*_StateTimer.IN:=TRUE;

IF _StateTimer.Q THEN
	_StateTimer.IN:=FALSE;
	M_StateComplete();
END_IF*)
END_METHOD

METHOD PROTECTED M_Resetting : BOOL
_StateTimer.IN:=TRUE;

IF _StateTimer.Q THEN
	_StateTimer.IN:=FALSE;
	M_StateComplete();
END_IF
END_METHOD

METHOD PROTECTED M_SetPackML : BOOL
_UnitMode(sName := 'Normal Operation', 
			dwSupportedStates := PACK_ML.State.All,
			dwAllowsLeavingFromStates := PACK_ML.State.Stopped 
											OR PACK_ML.State.Aborted 
											OR PACK_ML.State.Idle, 
			dwAllowsEnteringIntoStates := PACK_ML.State.Stopped
											OR PACK_ML.State.Aborted 
											OR PACK_ML.State.Idle, 
			eInitialState := PACK_ML.State.Idle,
			xActive := TRUE);
END_METHOD

METHOD PROTECTED M_Starting : BOOL
_StateTimer.IN:=TRUE;

IF _StateTimer.Q THEN
	_StateTimer.IN:=FALSE;
	M_StateComplete();
END_IF
END_METHOD

METHOD PROTECTED M_StateComplete : BOOL
_UnitMode.ActingStateCompleted();
END_METHOD

METHOD PROTECTED M_Stopped : BOOL
(*_StateTimer.IN:=TRUE;

IF _StateTimer.Q THEN
	_StateTimer.IN:=FALSE;
	M_StateComplete();
END_IF*)
END_METHOD

METHOD PROTECTED M_Stopping : BOOL
_StateTimer.IN:=TRUE;

IF _StateTimer.Q THEN
	_StateTimer.IN:=FALSE;
	M_StateComplete();
END_IF
END_METHOD

METHOD PROTECTED M_Suspended : BOOL
(*_StateTimer.IN:=TRUE;

IF _StateTimer.Q THEN
	_StateTimer.IN:=FALSE;
	M_StateComplete();
END_IF*)
END_METHOD

METHOD PROTECTED M_Suspending : BOOL
_StateTimer.IN:=TRUE;

IF _StateTimer.Q THEN
	_StateTimer.IN:=FALSE;
	M_StateComplete();
END_IF
END_METHOD

METHOD PROTECTED M_Unholding : BOOL
_StateTimer.IN:=TRUE;

IF _StateTimer.Q THEN
	_StateTimer.IN:=FALSE;
	M_StateComplete();
END_IF
END_METHOD

METHOD PROTECTED M_UnSuspending : BOOL
_StateTimer.IN:=TRUE;

IF _StateTimer.Q THEN
	_StateTimer.IN:=FALSE;
	M_StateComplete();
END_IF
END_METHOD

END_FUNCTION_BLOCK

// ---- FB/move/ParseMoveCmd.TcPOU
FUNCTION_BLOCK ParseMoveCmd
VAR_INPUT
	Command: STRING(GVL.COMMAND_LEN);
END_VAR
VAR_OUTPUT
	stCommand: ST_MoveCmd;
	Error: BOOL:= FALSE;
	ErrorDescription: STRING:='';
END_VAR
VAR
	_CmdParams: ARRAY [0..GVL.COMMAND_LEN] OF STRING;
END_VAR
VAR CONSTANT
	_MoveTypeD: STRING(3):='DIR';
	_MoveTypeL: STRING(3):='LIN';
	_MoveTypeC: STRING(3):='CIR';
	_ChangeTypeA: STRING(3):='ABS';
	_ChangeTypeR: STRING(3):='REL';
	_CoordSystemAcs: STRING(3):='ACS';
	_CoordSystemMcs: STRING(3):='MCS';
	_CoordSystemPc1: STRING(3):='PC1';
	_CoordSystemPc2: STRING(3):='PC2';
	_CoordSystemTcs: STRING(3):='TCS';
	_CoordSystemWcs: STRING(3):='WCS';
	_CoordSystemIcs: STRING(3):='ICS';
	_CoordTypeH: STRING(3):='LIT';
	_CoordTypeV: STRING(3):='VAR';
	_ArrayTypeS: STRING(3):='STO';
	_ArrayTypeV: STRING(3):='VIS';
	_ArrayTypeF: STRING(3):='FLG';
	_CircleModeBor: STRING(3):='BOR';
	_CircleModeCen: STRING(3):='CEN';
	_CircleModeRad: STRING(3):='RAD';
	_PathChoiceClw: STRING(3):='CLW';
	_PathChoiceCcw: STRING(3):='CCW';
END_VAR

// D is direct move. L is linear move. C is a circular move
// R is relative position. A is absolute position
// V is variable coordinated. H is a hardcoded coordinated
// S is stored position array. V is vision register array.
// D|L|C R|A Speed CoordSystem X0000.00 Y0000.00 Z0000.00 A0000.00 B0000.00 C0000.00 BOR|CEN|RAD CCW|CLW X0000.00 Y0000.00 Z0000.00 A0000.00 B0000.00 C0000.00
// 'D A 10 MCS H +0250.00 +0000.00 +0500.00 +0000.00 +0045.00 +0180.00'
// 'C R 10 MCS H +0250.00 +0000.00 +0500.00 +0000.00 +0045.00 +0180.00 BOR CLW H +0250.00 +0000.00 +0500.00 +0000.00 +0045.00 +0180.00'
// 'D A 10 MCS V S 25'
// 'D A 10 MCS V V 33'
// 'C R 10 MCS V S 2 BOR CLW V S 005'
// 'C R 10 MCS V S 003 BOR CLW V V 006'
// 'C R 10 MCS V S 015 BOR CLW H +0250.00 +0000.00 +0500.00 +0000.00 +0045.00 +0180.00'
// 'C R 10 MCS H 250.0 0.0 500.0 0.0 45.0 180.0 BOR CLW V V 22'

Error := FALSE;
ErrorDescription := '';

// split command string into commands
_CmdParams:=F_SplitCmd(Command:=Command);

//
IF _CmdParams[0] = _MoveTypeD THEN
	stCommand.MoveType := DUT_Command_MoveType.DirectMove;
ELSIF _CmdParams[0] = _MoveTypeL THEN
	stCommand.MoveType := DUT_Command_MoveType.LinearMove;
ELSIF _CmdParams[0] = _MoveTypeC THEN
	stCommand.MoveType := DUT_Command_MoveType.CircularMove;
ELSE
	Error := TRUE;
	ErrorDescription := 'Incorrect move type';
END_IF

//
IF _CmdParams[1] = _ChangeTypeR THEN
	stCommand.PositionType := DUT_Command_PositionType.RelativePosition;
ELSIF _CmdParams[1] = _ChangeTypeA THEN
	stCommand.PositionType := DUT_Command_PositionType.AbsolutePosition;
ELSE
	Error := TRUE;
	ErrorDescription := 'Incorrect position type';
END_IF

//
stCommand.Speed := STRING_TO_LREAL(_CmdParams[2]);

//
IF _CmdParams[3] = _CoordSystemAcs THEN
	stCommand.CoordSystem := DUT_CoordSystem.ACS;
ELSIF _CmdParams[3] = _CoordSystemMcs THEN
	stCommand.CoordSystem := DUT_CoordSystem.MCS;
ELSIF _CmdParams[3] = _CoordSystemPc1 THEN
	stCommand.CoordSystem := DUT_CoordSystem.UCS1;
ELSIF _CmdParams[3] = _CoordSystemPc2 THEN
	stCommand.CoordSystem := DUT_CoordSystem.UCS2;
ELSIF _CmdParams[3] = _CoordSystemTcs THEN
	stCommand.CoordSystem := DUT_CoordSystem.TCP;
// ELSIF _CmdParams[3] = _CoordSystemWcs THEN
// 	stCommand.CoordSystem := DUT_CoordSystem.WCS;
// ELSIF _CmdParams[3] = _CoordSystemIcs THEN
// 	stCommand.CoordSystem := DUT_CoordSystem.ICS;
ELSE
	Error := TRUE;
	ErrorDescription := 'Incorrect coordinate system type';
END_IF

//
IF _CmdParams[4] = _CoordTypeH THEN
	stCommand.CoordinateType := DUT_Command_CoordinateType.Literal;
ELSIF _CmdParams[4] = _CoordTypeV THEN
	stCommand.CoordinateType := DUT_Command_CoordinateType.Variable;
ELSE
	Error := TRUE;
	ErrorDescription := 'Incorrect coordinate type'; // TODO wow i need a better name for this... wtf was i thinking?
END_IF

//
CASE stCommand.CoordinateType OF 
// 'D A 010 MCS H +0250.00 +0000.00 +0500.00 +0000.00 +0045.00 +0180.00'
	DUT_Command_CoordinateType.Literal:
		stCommand.CoordRef.X := STRING_TO_LREAL(_CmdParams[5]);
		stCommand.CoordRef.Y := STRING_TO_LREAL(_CmdParams[6]);
		stCommand.CoordRef.Z := STRING_TO_LREAL(_CmdParams[7]);
		stCommand.CoordRef.A := STRING_TO_LREAL(_CmdParams[8]);
		stCommand.CoordRef.B := STRING_TO_LREAL(_CmdParams[9]);
		stCommand.CoordRef.C := STRING_TO_LREAL(_CmdParams[10]);
// 'D A 010 MCS V S 001'
	DUT_Command_CoordinateType.Variable:
		stCommand.ArrayIndex := STRING_TO_UINT(_CmdParams[6]);
		IF stCommand.ArrayIndex <= GVL.POS_ARR_END 
			AND stCommand.ArrayIndex >= GVL.POS_ARR_BEG THEN
				IF _CmdParams[5] = _ArrayTypeS THEN
					stCommand.ArrayType := DUT_Command_ArrayType.StoredPosition;
					stCommand.CoordRef := PersistentVars.StoredPositions[stCommand.ArrayIndex].Position;
				ELSIF _CmdParams[5] = _ArrayTypeV THEN
					stCommand.ArrayType := DUT_Command_ArrayType.VisionRegister;
					stCommand.CoordRef := PersistentVars.VisionRegisters[stCommand.ArrayIndex].Position;
				ELSE
					Error := TRUE;
					ErrorDescription := 'Incorrect array type';
				END_IF
		ELSE
			Error := TRUE;
			ErrorDescription := 'Array index out of bounds';
		END_IF
	
END_CASE

//
CASE stCommand.CoordinateType OF 
// 'C R 010 MCS H +0250.00 +0000.00 +0500.00 +0000.00 +0045.00 +0180.00 BOR CLW H +0250.00 +0000.00 +0500.00 +0000.00 +0045.00 +0180.00'
	DUT_Command_CoordinateType.Literal:
		IF _CmdParams[11] = _CircleModeBor THEN
			stCommand.CircleMode := MC_CIRC_MODE.mcCircModeBorder;
		ELSIF _CmdParams[11] = _CircleModeCen THEN
			stCommand.CircleMode := MC_CIRC_MODE.mcCircModeCenter;
		ELSIF _CmdParams[11] = _CircleModeRad THEN
			stCommand.CircleMode := MC_CIRC_MODE.mcCircModeRadius;
		ELSE
			Error := TRUE;
			ErrorDescription := 'Incorrect circle mode';
		END_IF
// 'C R 010 MCS V S 001 BOR CLW H +0250.00 +0000.00 +0500.00 +0000.00 +0045.00 +0180.00'
	DUT_Command_CoordinateType.Variable:
		IF _CmdParams[7] = _CircleModeBor THEN
			stCommand.CircleMode := MC_CIRC_MODE.mcCircModeBorder;
		ELSIF _CmdParams[7] = _CircleModeCen THEN
			stCommand.CircleMode := MC_CIRC_MODE.mcCircModeCenter;
		ELSIF _CmdParams[7] = _CircleModeRad THEN
			stCommand.CircleMode := MC_CIRC_MODE.mcCircModeRadius;
		ELSE
			Error := TRUE;
			ErrorDescription := 'Incorrect circle mode';
		END_IF
	
END_CASE

//
CASE stCommand.CoordinateType OF 
// 'C R 010 MCS H +0250.00 +0000.00 +0500.00 +0000.00 +0045.00 +0180.00 BOR CLW H +0250.00 +0000.00 +0500.00 +0000.00 +0045.00 +0180.00'
	DUT_Command_CoordinateType.Literal:
		IF _CmdParams[12] = _PathChoiceClw THEN
			stCommand.PathChoice := MC_CIRC_PATHCHOICE.mcCircPathChoiceClockwise;
		ELSIF _CmdParams[12] = _PathChoiceCcw THEN
			stCommand.PathChoice := MC_CIRC_PATHCHOICE.mcCircPathChoiceCounterClockwise;
		ELSE
			Error := TRUE;
			ErrorDescription := 'Incorrect circle direction';
		END_IF
		IF _CmdParams[13] = _CoordTypeH THEN
			stCommand.CircularCoordinateType := DUT_Command_CoordinateType.Literal;
		ELSIF _CmdParams[13] = _CoordTypeV THEN
			stCommand.CircularCoordinateType := DUT_Command_CoordinateType.Variable;
		ELSE
			Error := TRUE;
			ErrorDescription := 'Incorrect coordinate type'; // TODO yeah, this needs better naming. "coordinate type" does not fit.
		END_IF
// 'C R 010 MCS V S 001 BOR CLW H +0250.00 +0000.00 +0500.00 +0000.00 +0045.00 +0180.00'
	DUT_Command_CoordinateType.Variable:
		IF _CmdParams[8] = _PathChoiceClw THEN
			stCommand.PathChoice := MC_CIRC_PATHCHOICE.mcCircPathChoiceClockwise;
		ELSIF _CmdParams[8] = _PathChoiceCcw THEN
			stCommand.PathChoice := MC_CIRC_PATHCHOICE.mcCircPathChoiceCounterClockwise;
		ELSE
			Error := TRUE;
			ErrorDescription := 'Incorrect circle direction';
		END_IF
		IF _CmdParams[9] = _CoordTypeH THEN
			stCommand.CircularCoordinateType := DUT_Command_CoordinateType.Literal;
		ELSIF _CmdParams[9] = _CoordTypeV THEN
			stCommand.CircularCoordinateType := DUT_Command_CoordinateType.Variable;
		ELSE
			Error := TRUE;
			ErrorDescription := 'Incorrect coordinate type'; // TODO this naming "coordinate type" needs to go.
		END_IF
	
END_CASE

//
CASE stCommand.CircularCoordinateType OF 
	DUT_Command_CoordinateType.Literal:
		CASE stCommand.CoordinateType OF
// 'C R 010 MCS H +0250.00 +0000.00 +0500.00 +0000.00 +0045.00 +0180.00 BOR CLW H +0250.00 +0000.00 +0500.00 +0000.00 +0045.00 +0180.00'
			DUT_Command_CoordinateType.Literal:
				stCommand.CoordRef2.X := STRING_TO_LREAL(_CmdParams[14]);
				stCommand.CoordRef2.Y := STRING_TO_LREAL(_CmdParams[15]);
				stCommand.CoordRef2.Z := STRING_TO_LREAL(_CmdParams[16]);
				stCommand.CoordRef2.A := STRING_TO_LREAL(_CmdParams[17]);
				stCommand.CoordRef2.B := STRING_TO_LREAL(_CmdParams[18]);
				stCommand.CoordRef2.C := STRING_TO_LREAL(_CmdParams[19]);
// 'C R 010 MCS V S 001 BOR CLW H +0250.00 +0000.00 +0500.00 +0000.00 +0045.00 +0180.00'
			DUT_Command_CoordinateType.Variable:
				stCommand.CoordRef2.X := STRING_TO_LREAL(_CmdParams[10]);
				stCommand.CoordRef2.Y := STRING_TO_LREAL(_CmdParams[11]);
				stCommand.CoordRef2.Z := STRING_TO_LREAL(_CmdParams[12]);
				stCommand.CoordRef2.A := STRING_TO_LREAL(_CmdParams[13]);
				stCommand.CoordRef2.B := STRING_TO_LREAL(_CmdParams[14]);
				stCommand.CoordRef2.C := STRING_TO_LREAL(_CmdParams[15]);
				
		END_CASE
	
	DUT_Command_CoordinateType.Variable:
		CASE stCommand.CoordinateType OF
// 'C R 010 MCS H +0250.00 +0000.00 +0500.00 +0000.00 +0045.00 +0180.00 BOR CLW V V 001'
			DUT_Command_CoordinateType.Literal:
				stCommand.CircularArrayIndex := STRING_TO_UINT(_CmdParams[15]);
				IF stCommand.CircularArrayIndex <= GVL.POS_ARR_END 
					AND stCommand.CircularArrayIndex >= GVL.POS_ARR_BEG THEN
						IF _CmdParams[14] = _ArrayTypeS THEN
							stCommand.CircularArrayType := DUT_Command_ArrayType.StoredPosition;
							stCommand.CoordRef2 := PersistentVars.StoredPositions[stCommand.CircularArrayIndex].Position;
						ELSIF _CmdParams[14] = _ArrayTypeV THEN
							stCommand.CircularArrayType := DUT_Command_ArrayType.VisionRegister;
							stCommand.CoordRef2 := PersistentVars.VisionRegisters[stCommand.CircularArrayIndex].Position;
						ELSE
							Error := TRUE;
							ErrorDescription := 'Incorrect array type';
						END_IF
					
				ELSE
					Error:=TRUE;
					ErrorDescription := 'Array index out of bounds';
					
				END_IF
				
// 'C R 010 MCS V S 001 BOR CLW V V 001'
			DUT_Command_CoordinateType.Variable:
				stCommand.CircularArrayIndex := STRING_TO_UINT(_CmdParams[11]);
				IF stCommand.CircularArrayIndex <= GVL.POS_ARR_END 
					AND stCommand.CircularArrayIndex >= GVL.POS_ARR_BEG THEN
						IF _CmdParams[10] = _ArrayTypeS THEN
							stCommand.CircularArrayType := DUT_Command_ArrayType.StoredPosition;
							stCommand.CoordRef2 := PersistentVars.StoredPositions[stCommand.CircularArrayIndex].Position;
						ELSIF _CmdParams[10] = _ArrayTypeV THEN
							stCommand.CircularArrayType := DUT_Command_ArrayType.VisionRegister;
							stCommand.CoordRef2 := PersistentVars.VisionRegisters[stCommand.CircularArrayIndex].Position;
						ELSE
							Error:=TRUE;
							ErrorDescription := 'Incorrect array type';
						END_IF
					
				ELSE
					Error:=TRUE;
					ErrorDescription := 'Array index out of bounds';
				END_IF
				
		END_CASE
	
END_CASE

END_FUNCTION_BLOCK

// ---- FB/F_SplitCmd.TcPOU
FUNCTION F_SplitCmd : ARRAY [0..GVL.COMMAND_LEN] OF STRING
VAR_INPUT
    Command: STRING(GVL.COMMAND_LEN);
	Delimiter: STRING(1):=' ';
END_VAR
VAR
	_Command: STRING(GVL.COMMAND_LEN);
	_DelimPos: INT;
	_i, _j, _k: INT;
END_VAR
VAR CONSTANT
	_SpaceChar: STRING(1):=' ';
END_VAR

// grab a copy
// TODO do we need to do this? cant we just operate on the input?
_Command := Command;

// ex. 123 456 789 0 123 456 879 0
WHILE LEN(_Command) > 0  AND _i < GVL.COMMAND_LEN DO
	// find the delimiter
	_DelimPos := FIND(_Command, Delimiter);
	// don't copy empty commands
	IF _DelimPos > 1 THEN
		// copy the command into the array position
		F_SplitCmd[_i] := MID(STR:=_Command, LEN:=_DelimPos - 1, POS:=1);
		// trim the command off the front of the string
		_Command := DELETE(STR:=_Command, LEN:=_DelimPos, POS:=1);
		// increment the index and get ready for the next
		_i := _i + 1;
	ELSIF _DelimPos = 1 OR FIND(_Command, _SpaceChar) = 1 THEN
		// don't do anything with a stray delimiter or a space at the  start of the next command
		// trim the command off the space at the front of the string
		_Command := DELETE(STR:=_Command, LEN:=LEN(_SpaceChar), POS:=1);
	ELSIF _DelimPos = 0 AND LEN(_Command) > 0 THEN
		// copy the last command into the array position and return
		F_SplitCmd[_i] := MID(STR:=_Command, LEN:=LEN(_Command), POS:=1);
		// trim the command off the front of the string
		_Command := DELETE(STR:=_Command, LEN:=_DelimPos, POS:=1);
		// increment the index and get ready for the next
		_i := _i + 1;
		RETURN;
	ELSE
		RETURN;
	END_IF
END_WHILE

END_FUNCTION

// ---- FB/move/BuildMoveCmd.TcPOU
FUNCTION BuildMoveCmd : STRING(GVL.COMMAND_LEN);
VAR_INPUT
	stCommand: ST_MoveCmd;
END_VAR
VAR
	_Command : STRING(GVL.COMMAND_LEN);
END_VAR
VAR CONSTANT
	_Delimiter: STRING:=' ';
	_MoveTypeD: STRING(3):='DIR';
	_MoveTypeL: STRING(3):='LIN';
	_MoveTypeC: STRING(3):='CIR';
	_ChangeTypeA: STRING(3):='ABS';
	_ChangeTypeR: STRING(3):='REL';
	_CoordSystemAcs: STRING(3):='ACS';
	_CoordSystemMcs: STRING(3):='MCS';
	_CoordSystemPc1: STRING(3):='PC1';
	_CoordSystemPc2: STRING(3):='PC2';
	_CoordSystemTcs: STRING(3):='TCS';
	_CoordSystemWcs: STRING(3):='WCS';
	_CoordSystemIcs: STRING(3):='ICS';
	_CoordTypeH: STRING(3):='LIT';
	_CoordTypeV: STRING(3):='VAR';
	_ArrayTypeS: STRING(3):='STO';
	_ArrayTypeV: STRING(3):='VIS';
	_ArrayTypeF: STRING(3):='FLG';
	_CircleModeBor: STRING(3):='BOR';
	_CircleModeCen: STRING(3):='CEN';
	_CircleModeRad: STRING(3):='RAD';
	_PathChoiceClw: STRING(3):='CLW';
	_PathChoiceCcw: STRING(3):='CCW';
END_VAR

// D is direct move. L is linear move. C is a circular move
// R is relative position. A is absolute position
// V is variable coordinated. H is a hardcoded coordinated
// S is stored position array. V is vision register array.
// D|L|C R|A Speed CoordSystem X0000.00 Y0000.00 Z0000.00 A0000.00 B0000.00 C0000.00 BOR|CEN|RAD CCW|CLW X0000.00 Y0000.00 Z0000.00 A0000.00 B0000.00 C0000.00
// 'D A 010 MCS H +0250.00 +0000.00 +0500.00 +0000.00 +0045.00 +0180.00'
// 'C R 010 MCS H +0250.00 +0000.00 +0500.00 +0000.00 +0045.00 +0180.00 BOR CLW H +0250.00 +0000.00 +0500.00 +0000.00 +0045.00 +0180.00'
// 'D A 010 MCS V S 025'
// 'D A 010 MCS V V 033'
// 'C R 010 MCS V S 002 BOR CLW V S 005'
// 'C R 010 MCS V S 003 BOR CLW V V 006'
// 'C R 010 MCS V S 015 BOR CLW H +0250.00 +0000.00 +0500.00 +0000.00 +0045.00 +0180.00'
// 'C R 010 MCS H +0250.00 +0000.00 +0500.00 +0000.00 +0045.00 +0180.00 BOR CLW V V 022'

//
_Command := '';

//
CASE stCommand.MoveType OF
	DUT_Command_MoveType.DirectMove:
		F_AddElement(_Command, _Delimiter, _MoveTypeD);
	DUT_Command_MoveType.LinearMove:
		F_AddElement(_Command, _Delimiter, _MoveTypeL);
	DUT_Command_MoveType.CircularMove:
		F_AddElement(_Command, _Delimiter, _MoveTypeC);
END_CASE

//
CASE stCommand.PositionType OF
	DUT_Command_PositionType.AbsolutePosition:
		F_AddElement(_Command, _Delimiter, _ChangeTypeA);
	DUT_Command_PositionType.RelativePosition:
		F_AddElement(_Command, _Delimiter, _ChangeTypeR);
END_CASE

//
F_AddElement(_Command, _Delimiter, LREAL_TO_STRING(stCommand.Speed));

//
CASE stCommand.CoordSystem OF
	DUT_CoordSystem.ACS:
		F_AddElement(_Command, _Delimiter, _CoordSystemAcs);
	DUT_CoordSystem.MCS:
		F_AddElement(_Command, _Delimiter, _CoordSystemMcs);
	DUT_CoordSystem.UCS1:
		F_AddElement(_Command, _Delimiter, _CoordSystemPc1);
	DUT_CoordSystem.UCS2:
		F_AddElement(_Command, _Delimiter, _CoordSystemPc2);
	DUT_CoordSystem.TCP:
		F_AddElement(_Command, _Delimiter, _CoordSystemTcs);
// 	DUT_CoordSystem.WCS:
// 		F_AddElement(_Command, _Delimiter, _CoordSystemWcs);
// 	DUT_CoordSystem.ICS:
// 		F_AddElement(_Command, _Delimiter, _CoordSystemIcs);
END_CASE

